gfCNCPoint2[27573] = {X 365.5713, Y 5.1234, Z -3.8333, A 0.000, B 0.000, C 0.000 }
gfCNCPoint2[27574] = {X 365.9457, Y 5.5507, Z -3.8333, A 0.000, B 0.000, C 0.000 }
gfCNCPoint2[27575] = {X 367.0655, Y 6.9489, Z -3.8333, A 0.000, B 0.000, C 0.000 }
gfCNCPoint2[27576] = {X 368.0925, Y 8.4166, Z -3.8333, A 0.000, B 0.000, C 0.000 }
gfCNCPoint2[27577] = {X 369.3414, Y 10.5295, Z -3.8333, A 0.000, B 0.000, C 0.000 }
gfCNCPoint2[27578] = {X 370.3982, Y 12.7448, Z -3.8333, A 0.000, B 0.000, C 0.000 }
gfCNCPoint2[27579] = {X 371.2546, Y 15.0450, Z -3.8333, A 0.000, B 0.000, C 0.000 }
gfCNCPoint2[27580] = {X 371.9038, Y 17.4120, Z -3.8333, A 0.000, B 0.000, C 0.000 }
gfCNCPoint2[27581] = {X 372.3604, Y 19.8116, Z -3.8333, A 0.000, B 0.000, C 0.000 }
gfCNCPoint2[27582] = {X 372.6464, Y 22.2374, Z -3.8333, A 0.000, B 0.000, C 0.000 }
gfCNCPoint2[27583] = {X 372.7605, Y 24.6774, Z -3.8333, A 0.000, B 0.000, C 0.000 }
gfCNCPoint2[27584] = {X 372.7020, Y 27.1193, Z -3.8333, A 0.000, B 0.000, C 0.000 }
gfCNCPoint2[27585] = {X 372.4713, Y 29.5510, Z -3.8333, A 0.000, B 0.000, C 0.000 }
gfCNCPoint2[27586] = {X 372.0694, Y 31.9603, Z -3.8333, A 0.000, B 0.000, C 0.000 }
gfCNCPoint2[27587] = {X 371.4833, Y 34.3147, Z -3.8333, A 0.000, B 0.000, C 0.000 }
gfCNCPoint2[27588] = {X 370.6918, Y 36.6082, Z -3.8333, A 0.000, B 0.000, C 0.000 }
gfCNCPoint2[27589] = {X 369.7011, Y 38.8229, Z -3.8333, A 0.000, B 0.000, C 0.000 }
gfCNCPoint2[27590] = {X 368.5189, Y 40.9417, Z -3.8333, A 0.000, B 0.000, C 0.000 }
gfCNCPoint2[27591] = {X 367.1545, Y 42.9479, Z -3.8333, A 0.000, B 0.000, C 0.000 }
gfCNCPoint2[27592] = {X 367.0324, Y 43.1153, Z -3.8333, A 0.000, B 0.000, C 0.000 }
gfCNCPoint2[27593] = {X 366.9645, Y 43.2035, Z -3.8333, A 0.000, B 0.000, C 0.000 }
gfCNCPoint2[27594] = {X 366.3182, Y 43.9969, Z -3.8333, A 0.000, B 0.000, C 0.000 }
gfCNCPoint2[27595] = {X 364.8822, Y 45.6080, Z -3.8333, A 0.000, B 0.000, C 0.000 }
gfCNCPoint2[27596] = {X 363.3086, Y 47.0851, Z -3.8333, A 0.000, B 0.000, C 0.000 }
gfCNCPoint2[27597] = {X 361.6099, Y 48.4164, Z -3.8333, A 0.000, B 0.000, C 0.000 }
gfCNCPoint2[27598] = {X 359.7996, Y 49.5915, Z -3.8333, A 0.000, B 0.000, C 0.000 }
gfCNCPoint2[27599] = {X 357.8920, Y 50.6010, Z -3.8333, A 0.000, B 0.000, C 0.000 }
gfCNCPoint2[27600] = {X 357.4593, Y 50.8059, Z -3.8333, A 0.000, B 0.000, C 0.000 }
gfCNCPoint2[27601] = {X 355.4789, Y 51.5741, Z -3.8333, A 0.000, B 0.000, C 0.000 }
gfCNCPoint2[27602] = {X 353.4424, Y 52.1780, Z -3.8333, A 0.000, B 0.000, C 0.000 }
gfCNCPoint2[27603] = {X 351.3633, Y 52.6134, Z -3.8333, A 0.000, B 0.000, C 0.000 }
gfCNCPoint2[27604] = {X 349.2556, Y 52.8775, Z -3.8333, A 0.000, B 0.000, C 0.000 }
gfCNCPoint2[27605] = {X 347.1333, Y 52.9685, Z -3.8333, A 0.000, B 0.000, C 0.000 }
gfCNCPoint2[27606] = {X 344.8131, Y 52.9262, Z -3.8333, A 0.000, B 0.000, C 0.000 }
gfCNCPoint2[27607] = {X 342.5052, Y 52.6831, Z -3.8333, A 0.000, B 0.000, C 0.000 }
gfCNCPoint2[27608] = {X 340.2271, Y 52.2410, Z -3.8333, A 0.000, B 0.000, C 0.000 }
gfCNCPoint2[27609] = {X 337.9959, Y 51.6033, Z -3.8333, A 0.000, B 0.000, C 0.000 }
gfCNCPoint2[27610] = {X 335.8282, Y 50.7746, Z -3.8333, A 0.000, B 0.000, C 0.000 }
gfCNCPoint2[27611] = {X 333.7405, Y 49.7614, Z -3.8333, A 0.000, B 0.000, C 0.000 }
gfCNCPoint2[27612] = {X 332.8345, Y 49.2281, Z -3.8333, A 0.000, B 0.000, C 0.000 }
gfCNCPoint2[27613] = {X 331.9502, Y 48.6598, Z -3.8333, A 0.000, B 0.000, C 0.000 }
gfCNCPoint2[27614] = {X 331.3028, Y 48.2115, Z -3.8333, A 0.000, B 0.000, C 0.000 }
gfCNCPoint2[27615] = {X 330.6689, Y 47.7445, Z -3.8333, A 0.000, B 0.000, C 0.000 }
gfCNCPoint2[27616] = {X 329.2171, Y 49.6556, Z -3.8333, A 0.000, B 0.000, C 0.000 }
gfCNCPoint2[27617] = {X 328.8724, Y 49.3896, Z -3.8333, A 0.000, B 0.000, C 0.000 }
gfCNCPoint2[27618] = {X 328.5317, Y 49.1186, Z -3.8333, A 0.000, B 0.000, C 0.000 }
gfCNCPoint2[27619] = {X 328.1266, Y 49.0390, Z -3.8333, A 0.000, B 0.000, C 0.000 }
gfCNCPoint2[27620] = {X 327.7253, Y 48.9423, Z -3.8333, A 0.000, B 0.000, C 0.000 }
gfCNCPoint2[27621] = {X 328.4864, Y 49.2670, Z -3.8333, A 0.000, B 0.000, C 0.000 }
gfCNCPoint2[27622] = {X 329.2171, Y 49.6556, Z -3.8333, A 0.000, B 0.000, C 0.000 }
gfCNCPoint2[27623] = {X 330.6689, Y 47.7445, Z -3.8333, A 0.000, B 0.000, C 0.000 }
gfCNCPoint2[27624] = {X 330.0951, Y 47.2962, Z -3.8333, A 0.000, B 0.000, C 0.000 }
gfCNCPoint2[27625] = {X 329.5337, Y 46.8324, Z -3.8333, A 0.000, B 0.000, C 0.000 }
gfCNCPoint2[27626] = {X 328.9312, Y 46.7520, Z -3.8333, A 0.000, B 0.000, C 0.000 }
gfCNCPoint2[27627] = {X 328.3374, Y 46.6216, Z -3.8333, A 0.000, B 0.000, C 0.000 }
gfCNCPoint2[27628] = {X 327.9789, Y 46.5172, Z -3.8333, A 0.000, B 0.000, C 0.000 }
gfCNCPoint2[27629] = {X 327.6263, Y 46.3944, Z -3.8333, A 0.000, B 0.000, C 0.000 }
gfCNCPoint2[27630] = {X 326.7320, Y 45.9864, Z -3.8333, A 0.000, B 0.000, C 0.000 }
gfCNCPoint2[27631] = {X 325.9009, Y 45.4616, Z -3.8333, A 0.000, B 0.000, C 0.000 }
gfCNCPoint2[27632] = {X 325.1480, Y 44.8296, Z -3.8333, A 0.000, B 0.000, C 0.000 }
gfCNCPoint2[27633] = {X 324.5140, Y 44.2115, Z -3.8333, A 0.000, B 0.000, C 0.000 }
gfCNCPoint2[27634] = {X 324.0475, Y 43.7117, Z -3.8333, A 0.000, B 0.000, C 0.000 }
gfCNCPoint2[27635] = {X 323.6300, Y 43.1703, Z -3.8333, A 0.000, B 0.000, C 0.000 }
gfCNCPoint2[27636] = {X 319.6957, Y 45.9200, Z -3.8333, A 0.000, B 0.000, C 0.000 }
gfCNCPoint2[27637] = {X 319.4780, Y 45.5976, Z -3.8333, A 0.000, B 0.000, C 0.000 }
gfCNCPoint2[27638] = {X 319.2708, Y 45.2683, Z -3.8333, A 0.000, B 0.000, C 0.000 }
gfCNCPoint2[27639] = {X 319.2514, Y 45.5948, Z -3.8333, A 0.000, B 0.000, C 0.000 }
gfCNCPoint2[27640] = {X 319.2174, Y 45.9200, Z -3.8333, A 0.000, B 0.000, C 0.000 }
gfCNCPoint2[27641] = {X 319.6957, Y 45.9200, Z -3.8333, A 0.000, B 0.000, C 0.000 }
gfCNCPoint2[27642] = {X 321.6628, Y 44.5452, Z -3.8333, A 0.000, B 0.000, C 0.000 }
gfCNCPoint2[27643] = {X 321.4884, Y 44.2868, Z -3.8333, A 0.000, B 0.000, C 0.000 }
gfCNCPoint2[27644] = {X 321.3224, Y 44.0230, Z -3.8333, A 0.000, B 0.000, C 0.000 }
gfCNCPoint2[27645] = {X 320.6712, Y 42.7455, Z -3.8333, A 0.000, B 0.000, C 0.000 }
gfCNCPoint2[27646] = {X 320.2158, Y 41.3859, Z -3.8333, A 0.000, B 0.000, C 0.000 }
gfCNCPoint2[27647] = {X 319.9663, Y 39.9740, Z -3.8333, A 0.000, B 0.000, C 0.000 }
gfCNCPoint2[27648] = {X 319.9281, Y 38.5406, Z -3.8333, A 0.000, B 0.000, C 0.000 }
gfCNCPoint2[27649] = {X 320.1020, Y 37.1174, Z -3.8333, A 0.000, B 0.000, C 0.000 }
gfCNCPoint2[27650] = {X 320.4301, Y 35.8909, Z -3.8333, A 0.000, B 0.000, C 0.000 }
gfCNCPoint2[27651] = {X 320.9158, Y 34.7180, Z -3.8333, A 0.000, B 0.000, C 0.000 }
gfCNCPoint2[27652] = {X 321.5508, Y 33.6186, Z -3.8333, A 0.000, B 0.000, C 0.000 }
gfCNCPoint2[27653] = {X 324.1378, Y 29.7505, Z -3.8333, A 0.000, B 0.000, C 0.000 }
gfCNCPoint2[27654] = {X 320.1479, Y 27.0821, Z -3.8333, A 0.000, B 0.000, C 0.000 }
gfCNCPoint2[27655] = {X 321.8042, Y 24.6057, Z -3.8333, A 0.000, B 0.000, C 0.000 }
gfCNCPoint2[27656] = {X 321.9898, Y 24.3356, Z -3.8333, A 0.000, B 0.000, C 0.000 }
gfCNCPoint2[27657] = {X 322.1814, Y 24.0697, Z -3.8333, A 0.000, B 0.000, C 0.000 }
gfCNCPoint2[27658] = {X 321.5380, Y 23.0772, Z -3.8333, A 0.000, B 0.000, C 0.000 }
gfCNCPoint2[27659] = {X 320.9777, Y 22.0354, Z -3.8333, A 0.000, B 0.000, C 0.000 }
gfCNCPoint2[27660] = {X 320.1480, Y 20.3286, Z -3.8333, A 0.000, B 0.000, C 0.000 }
gfCNCPoint2[27661] = {X 320.1479, Y 27.0821, Z -3.8333, A 0.000, B 0.000, C 0.000 }
gfCNCPoint2[27662] = {X 322.1429, Y 28.4163, Z -3.8333, A 0.000, B 0.000, C 0.000 }
gfCNCPoint2[27663] = {X 323.7975, Y 25.9423, Z -3.8333, A 0.000, B 0.000, C 0.000 }
gfCNCPoint2[27664] = {X 324.5112, Y 24.9841, Z -3.8333, A 0.000, B 0.000, C 0.000 }
gfCNCPoint2[27665] = {X 325.3162, Y 24.1010, Z -3.8333, A 0.000, B 0.000, C 0.000 }
gfCNCPoint2[27666] = {X 324.4812, Y 23.1413, Z -3.8333, A 0.000, B 0.000, C 0.000 }
gfCNCPoint2[27667] = {X 323.7518, Y 22.0990, Z -3.8333, A 0.000, B 0.000, C 0.000 }
gfCNCPoint2[27668] = {X 323.1360, Y 20.9859, Z -3.8333, A 0.000, B 0.000, C 0.000 }
gfCNCPoint2[27669] = {X 319.6151, Y 13.7428, Z -3.8333, A 0.000, B 0.000, C 0.000 }
gfCNCPoint2[27670] = {X 319.4387, Y 13.3633, Z -3.8333, A 0.000, B 0.000, C 0.000 }
gfCNCPoint2[27671] = {X 319.2755, Y 12.9779, Z -3.8333, A 0.000, B 0.000, C 0.000 }
gfCNCPoint2[27672] = {X 319.2755, Y 13.0353, Z -3.8333, A 0.000, B 0.000, C 0.000 }
gfCNCPoint2[27673] = {X 319.1698, Y 14.2156, Z -3.8333, A 0.000, B 0.000, C 0.000 }
gfCNCPoint2[27674] = {X 318.8739, Y 15.3632, Z -3.8333, A 0.000, B 0.000, C 0.000 }
gfCNCPoint2[27675] = {X 318.3958, Y 16.4476, Z -3.8333, A 0.000, B 0.000, C 0.000 }
gfCNCPoint2[27676] = {X 317.7480, Y 17.4400, Z -3.8333, A 0.000, B 0.000, C 0.000 }
gfCNCPoint2[27677] = {X 317.7478, Y 36.6506, Z -3.8333, A 0.000, B 0.000, C 0.000 }
gfCNCPoint2[27678] = {X 318.1572, Y 35.1201, Z -3.8333, A 0.000, B 0.000, C 0.000 }
gfCNCPoint2[27679] = {X 318.7634, Y 33.6563, Z -3.8333, A 0.000, B 0.000, C 0.000 }
gfCNCPoint2[27680] = {X 319.5559, Y 32.2844, Z -3.8333, A 0.000, B 0.000, C 0.000 }
gfCNCPoint2[27681] = {X 322.1429, Y 28.4163, Z -3.8333, A 0.000, B 0.000, C 0.000 }
gfCNCPoint2[27682] = {X 324.1378, Y 29.7505, Z -3.8333, A 0.000, B 0.000, C 0.000 }
gfCNCPoint2[27683] = {X 325.7908, Y 27.2790, Z -3.8333, A 0.000, B 0.000, C 0.000 }
gfCNCPoint2[27684] = {X 326.3627, Y 26.5111, Z -3.8333, A 0.000, B 0.000, C 0.000 }
gfCNCPoint2[27685] = {X 327.0077, Y 25.8035, Z -3.8333, A 0.000, B 0.000, C 0.000 }
gfCNCPoint2[27686] = {X 328.0707, Y 24.8904, Z -3.8333, A 0.000, B 0.000, C 0.000 }
gfCNCPoint2[27687] = {X 329.2543, Y 24.1403, Z -3.8333, A 0.000, B 0.000, C 0.000 }
gfCNCPoint2[27688] = {X 328.0859, Y 23.3667, Z -3.8333, A 0.000, B 0.000, C 0.000 }
gfCNCPoint2[27689] = {X 327.0414, Y 22.4326, Z -3.8333, A 0.000, B 0.000, C 0.000 }
gfCNCPoint2[27690] = {X 326.3723, Y 21.6635, Z -3.8333, A 0.000, B 0.000, C 0.000 }
gfCNCPoint2[27691] = {X 325.7878, Y 20.8284, Z -3.8333, A 0.000, B 0.000, C 0.000 }
gfCNCPoint2[27692] = {X 325.2944, Y 19.9364, Z -3.8333, A 0.000, B 0.000, C 0.000 }
gfCNCPoint2[27693] = {X 321.7736, Y 12.6936, Z -3.8333, A 0.000, B 0.000, C 0.000 }
gfCNCPoint2[27694] = {X 321.6322, Y 12.3894, Z -3.8333, A 0.000, B 0.000, C 0.000 }
gfCNCPoint2[27695] = {X 321.5015, Y 12.0806, Z -3.8333, A 0.000, B 0.000, C 0.000 }
gfCNCPoint2[27696] = {X 321.1058, Y 10.8774, Z -3.8333, A 0.000, B 0.000, C 0.000 }
gfCNCPoint2[27697] = {X 320.8706, Y 9.6327, Z -3.8333, A 0.000, B 0.000, C 0.000 }
gfCNCPoint2[27698] = {X 320.7999, Y 8.3681, Z -3.8333, A 0.000, B 0.000, C 0.000 }
gfCNCPoint2[27699] = {X 320.8950, Y 7.1050, Z -3.8333, A 0.000, B 0.000, C 0.000 }
gfCNCPoint2[27700] = {X 298.7842, Y 7.1050, Z -3.8333, A 0.000, B 0.000, C 0.000 }
gfCNCPoint2[27701] = {X 298.7842, Y 9.5050, Z -3.8333, A 0.000, B 0.000, C 0.000 }
gfCNCPoint2[27702] = {X 297.8292, Y 9.5050, Z -3.8333, A 0.000, B 0.000, C 0.000 }
gfCNCPoint2[27703] = {X 298.1371, Y 10.4755, Z -3.8333, A 0.000, B 0.000, C 0.000 }
gfCNCPoint2[27704] = {X 298.3067, Y 11.4795, Z -3.8333, A 0.000, B 0.000, C 0.000 }
gfCNCPoint2[27705] = {X 298.4762, Y 10.4755, Z -3.8333, A 0.000, B 0.000, C 0.000 }
gfCNCPoint2[27706] = {X 298.7842, Y 9.5050, Z -3.8333, A 0.000, B 0.000, C 0.000 }
gfCNCPoint2[27707] = {X 298.7842, Y 7.1050, Z -3.8333, A 0.000, B 0.000, C 0.000 }
gfCNCPoint2[27708] = {X 207.3611, Y 7.1050, Z -3.8333, A 0.000, B 0.000, C 0.000 }
gfCNCPoint2[27709] = {X 207.3611, Y 11.9050, Z -3.8333, A 0.000, B 0.000, C 0.000 }
gfCNCPoint2[27710] = {X 205.8559, Y 11.9050, Z -3.8333, A 0.000, B 0.000, C 0.000 }
gfCNCPoint2[27711] = {X 206.6109, Y 13.3410, Z -3.8333, A 0.000, B 0.000, C 0.000 }
gfCNCPoint2[27712] = {X 207.2366, Y 14.8379, Z -3.8333, A 0.000, B 0.000, C 0.000 }
gfCNCPoint2[27713] = {X 207.7977, Y 16.7110, Z -3.8333, A 0.000, B 0.000, C 0.000 }
gfCNCPoint2[27714] = {X 208.1767, Y 18.6291, Z -3.8333, A 0.000, B 0.000, C 0.000 }
gfCNCPoint2[27715] = {X 208.3702, Y 20.5748, Z -3.8333, A 0.000, B 0.000, C 0.000 }
gfCNCPoint2[27716] = {X 208.3763, Y 22.5301, Z -3.8333, A 0.000, B 0.000, C 0.000 }
gfCNCPoint2[27717] = {X 208.1951, Y 24.4769, Z -3.8333, A 0.000, B 0.000, C 0.000 }
gfCNCPoint2[27718] = {X 207.8282, Y 26.3974, Z -3.8333, A 0.000, B 0.000, C 0.000 }
gfCNCPoint2[27719] = {X 207.3612, Y 28.0098, Z -3.8333, A 0.000, B 0.000, C 0.000 }
gfCNCPoint2[27720] = {X 206.7379, Y 29.5684, Z -3.8333, A 0.000, B 0.000, C 0.000 }
gfCNCPoint2[27721] = {X 205.9643, Y 31.0582, Z -3.8333, A 0.000, B 0.000, C 0.000 }
gfCNCPoint2[27722] = {X 206.0464, Y 31.2164, Z -3.8333, A 0.000, B 0.000, C 0.000 }
gfCNCPoint2[27723] = {X 206.1255, Y 31.3761, Z -3.8333, A 0.000, B 0.000, C 0.000 }
gfCNCPoint2[27724] = {X 208.8852, Y 37.0775, Z -3.8333, A 0.000, B 0.000, C 0.000 }
gfCNCPoint2[27725] = {X 208.8852, Y 18.1982, Z -3.8333, A 0.000, B 0.000, C 0.000 }
gfCNCPoint2[27726] = {X 208.2331, Y 17.0021, Z -3.8333, A 0.000, B 0.000, C 0.000 }
gfCNCPoint2[27727] = {X 207.7553, Y 15.7263, Z -3.8333, A 0.000, B 0.000, C 0.000 }
gfCNCPoint2[27728] = {X 207.4614, Y 14.3961, Z -3.8333, A 0.000, B 0.000, C 0.000 }
gfCNCPoint2[27729] = {X 207.3572, Y 13.0378, Z -3.8333, A 0.000, B 0.000, C 0.000 }
gfCNCPoint2[27730] = {X 207.3570, Y 12.1868, Z -3.8333, A 0.000, B 0.000, C 0.000 }
gfCNCPoint2[27731] = {X 207.3580, Y 12.0459, Z -3.8333, A 0.000, B 0.000, C 0.000 }
gfCNCPoint2[27732] = {X 207.3611, Y 11.9050, Z -3.8333, A 0.000, B 0.000, C 0.000 }
gfCNCPoint2[27733] = {X 207.3611, Y 9.5050, Z -3.8333, A 0.000, B 0.000, C 0.000 }
gfCNCPoint2[27734] = {X 200.9069, Y 9.5050, Z -3.8333, A 0.000, B 0.000, C 0.000 }
gfCNCPoint2[27735] = {X 201.9803, Y 10.6137, Z -3.8333, A 0.000, B 0.000, C 0.000 }
gfCNCPoint2[27736] = {X 202.9419, Y 11.8206, Z -3.8333, A 0.000, B 0.000, C 0.000 }
gfCNCPoint2[27737] = {X 203.7829, Y 13.1145, Z -3.8333, A 0.000, B 0.000, C 0.000 }
gfCNCPoint2[27738] = {X 204.4363, Y 14.3564, Z -3.8333, A 0.000, B 0.000, C 0.000 }
gfCNCPoint2[27739] = {X 204.9784, Y 15.6507, Z -3.8333, A 0.000, B 0.000, C 0.000 }
gfCNCPoint2[27740] = {X 205.5510, Y 17.6374, Z -3.8333, A 0.000, B 0.000, C 0.000 }
gfCNCPoint2[27741] = {X 205.8919, Y 19.6767, Z -3.8333, A 0.000, B 0.000, C 0.000 }
gfCNCPoint2[27742] = {X 205.9964, Y 21.7416, Z -3.8333, A 0.000, B 0.000, C 0.000 }
gfCNCPoint2[27743] = {X 205.8631, Y 23.8049, Z -3.8333, A 0.000, B 0.000, C 0.000 }
gfCNCPoint2[27744] = {X 205.4940, Y 25.8393, Z -3.8333, A 0.000, B 0.000, C 0.000 }
gfCNCPoint2[27745] = {X 205.0929, Y 27.2255, Z -3.8333, A 0.000, B 0.000, C 0.000 }
gfCNCPoint2[27746] = {X 204.5574, Y 28.5655, Z -3.8333, A 0.000, B 0.000, C 0.000 }
gfCNCPoint2[27747] = {X 203.8927, Y 29.8464, Z -3.8333, A 0.000, B 0.000, C 0.000 }
gfCNCPoint2[27748] = {X 203.1052, Y 31.0557, Z -3.8333, A 0.000, B 0.000, C 0.000 }
gfCNCPoint2[27749] = {X 203.5732, Y 31.7148, Z -3.8333, A 0.000, B 0.000, C 0.000 }
gfCNCPoint2[27750] = {X 203.9653, Y 32.4217, Z -3.8333, A 0.000, B 0.000, C 0.000 }
gfCNCPoint2[27751] = {X 206.9865, Y 38.6634, Z -3.8333, A 0.000, B 0.000, C 0.000 }
gfCNCPoint2[27752] = {X 207.4240, Y 39.8017, Z -3.8333, A 0.000, B 0.000, C 0.000 }
gfCNCPoint2[27753] = {X 207.6653, Y 40.9971, Z -3.8333, A 0.000, B 0.000, C 0.000 }
gfCNCPoint2[27754] = {X 207.7038, Y 42.2159, Z -3.8333, A 0.000, B 0.000, C 0.000 }
gfCNCPoint2[27755] = {X 207.5382, Y 43.4241, Z -3.8333, A 0.000, B 0.000, C 0.000 }
gfCNCPoint2[27756] = {X 207.1733, Y 44.5877, Z -3.8333, A 0.000, B 0.000, C 0.000 }
gfCNCPoint2[27757] = {X 206.6193, Y 45.6741, Z -3.8333, A 0.000, B 0.000, C 0.000 }
gfCNCPoint2[27758] = {X 205.8917, Y 46.6527, Z -3.8333, A 0.000, B 0.000, C 0.000 }
gfCNCPoint2[27759] = {X 205.0110, Y 47.4962, Z -3.8333, A 0.000, B 0.000, C 0.000 }
gfCNCPoint2[27760] = {X 204.4738, Y 47.9305, Z -3.8333, A 0.000, B 0.000, C 0.000 }
gfCNCPoint2[27761] = {X 203.5892, Y 48.5431, Z -3.8333, A 0.000, B 0.000, C 0.000 }
gfCNCPoint2[27762] = {X 202.6241, Y 49.0188, Z -3.8333, A 0.000, B 0.000, C 0.000 }
gfCNCPoint2[27763] = {X 201.4895, Y 49.3730, Z -3.8333, A 0.000, B 0.000, C 0.000 }
gfCNCPoint2[27764] = {X 200.3125, Y 49.5382, Z -3.8333, A 0.000, B 0.000, C 0.000 }
gfCNCPoint2[27765] = {X 199.1243, Y 49.5100, Z -3.8333, A 0.000, B 0.000, C 0.000 }
gfCNCPoint2[27766] = {X 196.8333, Y 50.6067, Z -3.8333, A 0.000, B 0.000, C 0.000 }
gfCNCPoint2[27767] = {X 194.4618, Y 51.5162, Z -3.8333, A 0.000, B 0.000, C 0.000 }
gfCNCPoint2[27768] = {X 192.0250, Y 52.2327, Z -3.8333, A 0.000, B 0.000, C 0.000 }
gfCNCPoint2[27769] = {X 190.7221, Y 52.5183, Z -3.8333, A 0.000, B 0.000, C 0.000 }
gfCNCPoint2[27770] = {X 189.4061, Y 52.7356, Z -3.8333, A 0.000, B 0.000, C 0.000 }
gfCNCPoint2[27771] = {X 189.9005, Y 53.9113, Z -3.8333, A 0.000, B 0.000, C 0.000 }
gfCNCPoint2[27772] = {X 190.2683, Y 55.1326, Z -3.8333, A 0.000, B 0.000, C 0.000 }
gfCNCPoint2[27773] = {X 190.5269, Y 56.5560, Z -3.8333, A 0.000, B 0.000, C 0.000 }
gfCNCPoint2[27774] = {X 190.6135, Y 58.0000, Z -3.8333, A 0.000, B 0.000, C 0.000 }
gfCNCPoint2[27775] = {X 190.6132, Y 58.8767, Z -3.8333, A 0.000, B 0.000, C 0.000 }
gfCNCPoint2[27776] = {X 208.6252, Y 78.5345, Z -3.8333, A 0.000, B 0.000, C 0.000 }
gfCNCPoint2[27777] = {X 212.1642, Y 75.2918, Z -3.8333, A 0.000, B 0.000, C 0.000 }
gfCNCPoint2[27778] = {X 215.1994, Y 78.6043, Z -3.8333, A 0.000, B 0.000, C 0.000 }
gfCNCPoint2[27779] = {X 218.3280, Y 76.5999, Z -3.8333, A 0.000, B 0.000, C 0.000 }
gfCNCPoint2[27780] = {X 216.9962, Y 76.0772, Z -3.8333, A 0.000, B 0.000, C 0.000 }
gfCNCPoint2[27781] = {X 216.3765, Y 75.8848, Z -3.8333, A 0.000, B 0.000, C 0.000 }
gfCNCPoint2[27782] = {X 215.7328, Y 75.8035, Z -3.8333, A 0.000, B 0.000, C 0.000 }
gfCNCPoint2[27783] = {X 213.9348, Y 75.6432, Z -3.8333, A 0.000, B 0.000, C 0.000 }
gfCNCPoint2[27784] = {X 212.1642, Y 75.2918, Z -3.8333, A 0.000, B 0.000, C 0.000 }
gfCNCPoint2[27785] = {X 210.3947, Y 76.9131, Z -3.8333, A 0.000, B 0.000, C 0.000 }
gfCNCPoint2[27786] = {X 214.7939, Y 81.7143, Z -3.8333, A 0.000, B 0.000, C 0.000 }
gfCNCPoint2[27787] = {X 223.5827, Y 76.0838, Z -3.8333, A 0.000, B 0.000, C 0.000 }
gfCNCPoint2[27788] = {X 217.8854, Y 73.8480, Z -3.8333, A 0.000, B 0.000, C 0.000 }
gfCNCPoint2[27789] = {X 216.8722, Y 73.5366, Z -3.8333, A 0.000, B 0.000, C 0.000 }
gfCNCPoint2[27790] = {X 215.8204, Y 73.4051, Z -3.8333, A 0.000, B 0.000, C 0.000 }
gfCNCPoint2[27791] = {X 214.2768, Y 73.2676, Z -3.8333, A 0.000, B 0.000, C 0.000 }
gfCNCPoint2[27792] = {X 212.7566, Y 72.9660, Z -3.8333, A 0.000, B 0.000, C 0.000 }
gfCNCPoint2[27793] = {X 211.1575, Y 72.4584, Z -3.8333, A 0.000, B 0.000, C 0.000 }
gfCNCPoint2[27794] = {X 209.6279, Y 71.7692, Z -3.8333, A 0.000, B 0.000, C 0.000 }
gfCNCPoint2[27795] = {X 208.1882, Y 70.9078, Z -3.8333, A 0.000, B 0.000, C 0.000 }
gfCNCPoint2[27796] = {X 206.8579, Y 69.8855, Z -3.8333, A 0.000, B 0.000, C 0.000 }
gfCNCPoint2[27797] = {X 205.6547, Y 68.7163, Z -3.8333, A 0.000, B 0.000, C 0.000 }
gfCNCPoint2[27798] = {X 204.5949, Y 67.4157, Z -3.8333, A 0.000, B 0.000, C 0.000 }
gfCNCPoint2[27799] = {X 203.6926, Y 66.0013, Z -3.8333, A 0.000, B 0.000, C 0.000 }
gfCNCPoint2[27800] = {X 202.9600, Y 64.4920, Z -3.8333, A 0.000, B 0.000, C 0.000 }
gfCNCPoint2[27801] = {X 202.4068, Y 62.9081, Z -3.8333, A 0.000, B 0.000, C 0.000 }
gfCNCPoint2[27802] = {X 202.0406, Y 61.2709, Z -3.8333, A 0.000, B 0.000, C 0.000 }
gfCNCPoint2[27803] = {X 199.6721, Y 61.6582, Z -3.8333, A 0.000, B 0.000, C 0.000 }
gfCNCPoint2[27804] = {X 199.5095, Y 60.3402, Z -3.8333, A 0.000, B 0.000, C 0.000 }
gfCNCPoint2[27805] = {X 199.4510, Y 59.0136, Z -3.8333, A 0.000, B 0.000, C 0.000 }
gfCNCPoint2[27806] = {X 199.4508, Y 58.0000, Z -3.8333, A 0.000, B 0.000, C 0.000 }
gfCNCPoint2[27807] = {X 199.5412, Y 56.2556, Z -3.8333, A 0.000, B 0.000, C 0.000 }
gfCNCPoint2[27808] = {X 199.8114, Y 54.5298, Z -3.8333, A 0.000, B 0.000, C 0.000 }
gfCNCPoint2[27809] = {X 197.5977, Y 55.4810, Z -3.8333, A 0.000, B 0.000, C 0.000 }
gfCNCPoint2[27810] = {X 195.3260, Y 56.2839, Z -3.8333, A 0.000, B 0.000, C 0.000 }
gfCNCPoint2[27811] = {X 195.3578, Y 56.6300, Z -3.8333, A 0.000, B 0.000, C 0.000 }
gfCNCPoint2[27812] = {X 195.3825, Y 56.9766, Z -3.8333, A 0.000, B 0.000, C 0.000 }
gfCNCPoint2[27813] = {X 199.6721, Y 61.6582, Z -3.8333, A 0.000, B 0.000, C 0.000 }
gfCNCPoint2[27814] = {X 202.0406, Y 61.2709, Z -3.8333, A 0.000, B 0.000, C 0.000 }
gfCNCPoint2[27815] = {X 201.9013, Y 60.1428, Z -3.8333, A 0.000, B 0.000, C 0.000 }
gfCNCPoint2[27816] = {X 201.8510, Y 59.0073, Z -3.8333, A 0.000, B 0.000, C 0.000 }
gfCNCPoint2[27817] = {X 201.8508, Y 58.0000, Z -3.8333, A 0.000, B 0.000, C 0.000 }
gfCNCPoint2[27818] = {X 201.9283, Y 56.5036, Z -3.8333, A 0.000, B 0.000, C 0.000 }
gfCNCPoint2[27819] = {X 202.1601, Y 55.0232, Z -3.8333, A 0.000, B 0.000, C 0.000 }
gfCNCPoint2[27820] = {X 202.4969, Y 53.7230, Z -3.8333, A 0.000, B 0.000, C 0.000 }
gfCNCPoint2[27821] = {X 202.9527, Y 52.4596, Z -3.8333, A 0.000, B 0.000, C 0.000 }
gfCNCPoint2[27822] = {X 203.5236, Y 51.2439, Z -3.8333, A 0.000, B 0.000, C 0.000 }
gfCNCPoint2[27823] = {X 202.2637, Y 51.6554, Z -3.8333, A 0.000, B 0.000, C 0.000 }
gfCNCPoint2[27824] = {X 200.9594, Y 51.8913, Z -3.8333, A 0.000, B 0.000, C 0.000 }
gfCNCPoint2[27825] = {X 199.6352, Y 51.9470, Z -3.8333, A 0.000, B 0.000, C 0.000 }
gfCNCPoint2[27826] = {X 199.2148, Y 52.1550, Z -3.8333, A 0.000, B 0.000, C 0.000 }
gfCNCPoint2[27827] = {X 198.7916, Y 52.3572, Z -3.8333, A 0.000, B 0.000, C 0.000 }
gfCNCPoint2[27828] = {X 196.7764, Y 53.2250, Z -3.8333, A 0.000, B 0.000, C 0.000 }
gfCNCPoint2[27829] = {X 194.7096, Y 53.9612, Z -3.8333, A 0.000, B 0.000, C 0.000 }
gfCNCPoint2[27830] = {X 192.5997, Y 54.5629, Z -3.8333, A 0.000, B 0.000, C 0.000 }
gfCNCPoint2[27831] = {X 192.9063, Y 56.2411, Z -3.8333, A 0.000, B 0.000, C 0.000 }
gfCNCPoint2[27832] = {X 193.0134, Y 57.9437, Z -3.8333, A 0.000, B 0.000, C 0.000 }
gfCNCPoint2[27833] = {X 210.3947, Y 76.9131, Z -3.8333, A 0.000, B 0.000, C 0.000 }
gfCNCPoint2[27834] = {X 208.6252, Y 78.5345, Z -3.8333, A 0.000, B 0.000, C 0.000 }
gfCNCPoint2[27835] = {X 214.3884, Y 84.8243, Z -3.8333, A 0.000, B 0.000, C 0.000 }
gfCNCPoint2[27836] = {X 228.8373, Y 75.5678, Z -3.8333, A 0.000, B 0.000, C 0.000 }
gfCNCPoint2[27837] = {X 218.7726, Y 71.6180, Z -3.8333, A 0.000, B 0.000, C 0.000 }
gfCNCPoint2[27838] = {X 217.8432, Y 71.3042, Z -3.8333, A 0.000, B 0.000, C 0.000 }
gfCNCPoint2[27839] = {X 216.8839, Y 71.0995, Z -3.8333, A 0.000, B 0.000, C 0.000 }
gfCNCPoint2[27840] = {X 215.9073, Y 71.0066, Z -3.8333, A 0.000, B 0.000, C 0.000 }
gfCNCPoint2[27841] = {X 214.2374, Y 70.8313, Z -3.8333, A 0.000, B 0.000, C 0.000 }
gfCNCPoint2[27842] = {X 212.6079, Y 70.4261, Z -3.8333, A 0.000, B 0.000, C 0.000 }
gfCNCPoint2[27843] = {X 211.0503, Y 69.7988, Z -3.8333, A 0.000, B 0.000, C 0.000 }
gfCNCPoint2[27844] = {X 209.5948, Y 68.9617, Z -3.8333, A 0.000, B 0.000, C 0.000 }
gfCNCPoint2[27845] = {X 208.2694, Y 67.9308, Z -3.8333, A 0.000, B 0.000, C 0.000 }
gfCNCPoint2[27846] = {X 207.0998, Y 66.7260, Z -3.8333, A 0.000, B 0.000, C 0.000 }
gfCNCPoint2[27847] = {X 206.1085, Y 65.3707, Z -3.8333, A 0.000, B 0.000, C 0.000 }
gfCNCPoint2[27848] = {X 205.3147, Y 63.8911, Z -3.8333, A 0.000, B 0.000, C 0.000 }
gfCNCPoint2[27849] = {X 204.7338, Y 62.3157, Z -3.8333, A 0.000, B 0.000, C 0.000 }
gfCNCPoint2[27850] = {X 204.3769, Y 60.6749, Z -3.8333, A 0.000, B 0.000, C 0.000 }
gfCNCPoint2[27851] = {X 204.2510, Y 59.0005, Z -3.8333, A 0.000, B 0.000, C 0.000 }
gfCNCPoint2[27852] = {X 204.2508, Y 58.0000, Z -3.8333, A 0.000, B 0.000, C 0.000 }
gfCNCPoint2[27853] = {X 204.3397, Y 56.5376, Z -3.8333, A 0.000, B 0.000, C 0.000 }
gfCNCPoint2[27854] = {X 204.6049, Y 55.0967, Z -3.8333, A 0.000, B 0.000, C 0.000 }
gfCNCPoint2[27855] = {X 205.0426, Y 53.6986, Z -3.8333, A 0.000, B 0.000, C 0.000 }
gfCNCPoint2[27856] = {X 205.6463, Y 52.3637, Z -3.8333, A 0.000, B 0.000, C 0.000 }
gfCNCPoint2[27857] = {X 206.5298, Y 50.9383, Z -3.8333, A 0.000, B 0.000, C 0.000 }
gfCNCPoint2[27858] = {X 207.6022, Y 49.6491, Z -3.8333, A 0.000, B 0.000, C 0.000 }
gfCNCPoint2[27859] = {X 208.8428, Y 48.5208, Z -3.8333, A 0.000, B 0.000, C 0.000 }
gfCNCPoint2[27860] = {X 210.2277, Y 47.5751, Z -3.8333, A 0.000, B 0.000, C 0.000 }
gfCNCPoint2[27861] = {X 209.8801, Y 46.3328, Z -3.8333, A 0.000, B 0.000, C 0.000 }
gfCNCPoint2[27862] = {X 209.7572, Y 45.0487, Z -3.8333, A 0.000, B 0.000, C 0.000 }
gfCNCPoint2[27863] = {X 209.7570, Y 44.1967, Z -3.8333, A 0.000, B 0.000, C 0.000 }
gfCNCPoint2[27864] = {X 209.8559, Y 43.0066, Z -3.8333, A 0.000, B 0.000, C 0.000 }
gfCNCPoint2[27865] = {X 210.1498, Y 41.8492, Z -3.8333, A 0.000, B 0.000, C 0.000 }
gfCNCPoint2[27866] = {X 210.6306, Y 40.7561, Z -3.8333, A 0.000, B 0.000, C 0.000 }
gfCNCPoint2[27867] = {X 211.2852, Y 39.7574, Z -3.8333, A 0.000, B 0.000, C 0.000 }
gfCNCPoint2[27868] = {X 211.2852, Y 37.0775, Z -3.8333, A 0.000, B 0.000, C 0.000 }
gfCNCPoint2[27869] = {X 211.2849, Y 17.4403, Z -3.8333, A 0.000, B 0.000, C 0.000 }
gfCNCPoint2[27870] = {X 210.6364, Y 16.4465, Z -3.8333, A 0.000, B 0.000, C 0.000 }
gfCNCPoint2[27871] = {X 210.1579, Y 15.3605, Z -3.8333, A 0.000, B 0.000, C 0.000 }
gfCNCPoint2[27872] = {X 209.8622, Y 14.2112, Z -3.8333, A 0.000, B 0.000, C 0.000 }
gfCNCPoint2[27873] = {X 209.7572, Y 13.0291, Z -3.8333, A 0.000, B 0.000, C 0.000 }
gfCNCPoint2[27874] = {X 209.7570, Y 12.1868, Z -3.8333, A 0.000, B 0.000, C 0.000 }
gfCNCPoint2[27875] = {X 209.7578, Y 12.0808, Z -3.8333, A 0.000, B 0.000, C 0.000 }
gfCNCPoint2[27876] = {X 209.7601, Y 11.9749, Z -3.8333, A 0.000, B 0.000, C 0.000 }
gfCNCPoint2[27877] = {X 209.9068, Y 10.7177, Z -3.8333, A 0.000, B 0.000, C 0.000 }
gfCNCPoint2[27878] = {X 210.2690, Y 9.5050, Z -3.8333, A 0.000, B 0.000, C 0.000 }
gfCNCPoint2[27879] = {X 207.3611, Y 9.5050, Z -3.8333, A 0.000, B 0.000, C 0.000 }
gfCNCPoint2[27880] = {X 207.3611, Y 7.1050, Z -3.8333, A 0.000, B 0.000, C 0.000 }
gfCNCPoint2[27881] = {X 191.1443, Y 7.1050, Z -3.8333, A 0.000, B 0.000, C 0.000 }
gfCNCPoint2[27882] = {X 193.1012, Y 7.6483, Z -3.8333, A 0.000, B 0.000, C 0.000 }
gfCNCPoint2[27883] = {X 194.9845, Y 8.4084, Z -3.8333, A 0.000, B 0.000, C 0.000 }
gfCNCPoint2[27884] = {X 196.7702, Y 9.3758, Z -3.8333, A 0.000, B 0.000, C 0.000 }
gfCNCPoint2[27885] = {X 198.4355, Y 10.5381, Z -3.8333, A 0.000, B 0.000, C 0.000 }
gfCNCPoint2[27886] = {X 198.8575, Y 10.8885, Z -3.8333, A 0.000, B 0.000, C 0.000 }
gfCNCPoint2[27887] = {X 199.2650, Y 11.2555, Z -3.8333, A 0.000, B 0.000, C 0.000 }
gfCNCPoint2[27888] = {X 200.3500, Y 12.3982, Z -3.8333, A 0.000, B 0.000, C 0.000 }
gfCNCPoint2[27889] = {X 201.2956, Y 13.6586, Z -3.8333, A 0.000, B 0.000, C 0.000 }
gfCNCPoint2[27890] = {X 202.0892, Y 15.0198, Z -3.8333, A 0.000, B 0.000, C 0.000 }
gfCNCPoint2[27891] = {X 202.7202, Y 16.4636, Z -3.8333, A 0.000, B 0.000, C 0.000 }
gfCNCPoint2[27892] = {X 203.2139, Y 18.1834, Z -3.8333, A 0.000, B 0.000, C 0.000 }
gfCNCPoint2[27893] = {X 203.5072, Y 19.9484, Z -3.8333, A 0.000, B 0.000, C 0.000 }
gfCNCPoint2[27894] = {X 203.5963, Y 21.7354, Z -3.8333, A 0.000, B 0.000, C 0.000 }
gfCNCPoint2[27895] = {X 203.4800, Y 23.5208, Z -3.8333, A 0.000, B 0.000, C 0.000 }
gfCNCPoint2[27896] = {X 203.1598, Y 25.2812, Z -3.8333, A 0.000, B 0.000, C 0.000 }
gfCNCPoint2[27897] = {X 202.7594, Y 26.6265, Z -3.8333, A 0.000, B 0.000, C 0.000 }
gfCNCPoint2[27898] = {X 202.2078, Y 27.9173, Z -3.8333, A 0.000, B 0.000, C 0.000 }
gfCNCPoint2[27899] = {X 201.5122, Y 29.1365, Z -3.8333, A 0.000, B 0.000, C 0.000 }
gfCNCPoint2[27900] = {X 200.6817, Y 30.2681, Z -3.8333, A 0.000, B 0.000, C 0.000 }
gfCNCPoint2[27901] = {X 199.7272, Y 31.2973, Z -3.8333, A 0.000, B 0.000, C 0.000 }
gfCNCPoint2[27902] = {X 200.5668, Y 31.8698, Z -3.8333, A 0.000, B 0.000, C 0.000 }
gfCNCPoint2[27903] = {X 201.2695, Y 32.6038, Z -3.8333, A 0.000, B 0.000, C 0.000 }
gfCNCPoint2[27904] = {X 201.8050, Y 33.4674, Z -3.8333, A 0.000, B 0.000, C 0.000 }
gfCNCPoint2[27905] = {X 204.8262, Y 39.7091, Z -3.8333, A 0.000, B 0.000, C 0.000 }
gfCNCPoint2[27906] = {X 205.1508, Y 40.5847, Z -3.8333, A 0.000, B 0.000, C 0.000 }
gfCNCPoint2[27907] = {X 205.3026, Y 41.5062, Z -3.8333, A 0.000, B 0.000, C 0.000 }
gfCNCPoint2[27908] = {X 205.2761, Y 42.4397, Z -3.8333, A 0.000, B 0.000, C 0.000 }
gfCNCPoint2[27909] = {X 205.0723, Y 43.3511, Z -3.8333, A 0.000, B 0.000, C 0.000 }
gfCNCPoint2[27910] = {X 204.6986, Y 44.2070, Z -3.8333, A 0.000, B 0.000, C 0.000 }
gfCNCPoint2[27911] = {X 204.1687, Y 44.9760, Z -3.8333, A 0.000, B 0.000, C 0.000 }
gfCNCPoint2[27912] = {X 203.5020, Y 45.6299, Z -3.8333, A 0.000, B 0.000, C 0.000 }
gfCNCPoint2[27913] = {X 202.9657, Y 46.0636, Z -3.8333, A 0.000, B 0.000, C 0.000 }
gfCNCPoint2[27914] = {X 202.2136, Y 46.5639, Z -3.8333, A 0.000, B 0.000, C 0.000 }
gfCNCPoint2[27915] = {X 201.3824, Y 46.9175, Z -3.8333, A 0.000, B 0.000, C 0.000 }
gfCNCPoint2[27916] = {X 200.5003, Y 47.1123, Z -3.8333, A 0.000, B 0.000, C 0.000 }
gfCNCPoint2[27917] = {X 199.5975, Y 47.1416, Z -3.8333, A 0.000, B 0.000, C 0.000 }
gfCNCPoint2[27918] = {X 198.7046, Y 47.0045, Z -3.8333, A 0.000, B 0.000, C 0.000 }
gfCNCPoint2[27919] = {X 196.3903, Y 48.1789, Z -3.8333, A 0.000, B 0.000, C 0.000 }
gfCNCPoint2[27920] = {X 193.9811, Y 49.1437, Z -3.8333, A 0.000, B 0.000, C 0.000 }
gfCNCPoint2[27921] = {X 191.4959, Y 49.8913, Z -3.8333, A 0.000, B 0.000, C 0.000 }
gfCNCPoint2[27922] = {X 190.2926, Y 50.1569, Z -3.8333, A 0.000, B 0.000, C 0.000 }
gfCNCPoint2[27923] = {X 189.0769, Y 50.3583, Z -3.8333, A 0.000, B 0.000, C 0.000 }
gfCNCPoint2[27924] = {X 186.8985, Y 50.5559, Z -3.8333, A 0.000, B 0.000, C 0.000 }
gfCNCPoint2[27925] = {X 184.7112, Y 50.5476, Z -3.8333, A 0.000, B 0.000, C 0.000 }
gfCNCPoint2[27926] = {X 184.7356, Y 50.0682, Z -3.8333, A 0.000, B 0.000, C 0.000 }
gfCNCPoint2[27927] = {X 183.1153, Y 49.9273, Z -3.8333, A 0.000, B 0.000, C 0.000 }
gfCNCPoint2[27928] = {X 181.5093, Y 49.6709, Z -3.8333, A 0.000, B 0.000, C 0.000 }
gfCNCPoint2[27929] = {X 179.6141, Y 49.1972, Z -3.8333, A 0.000, B 0.000, C 0.000 }
gfCNCPoint2[27930] = {X 177.7853, Y 48.5105, Z -3.8333, A 0.000, B 0.000, C 0.000 }
gfCNCPoint2[27931] = {X 176.0466, Y 47.6200, Z -3.8333, A 0.000, B 0.000, C 0.000 }
gfCNCPoint2[27932] = {X 174.4207, Y 46.5371, Z -3.8333, A 0.000, B 0.000, C 0.000 }
gfCNCPoint2[27933] = {X 173.1806, Y 45.4904, Z -3.8333, A 0.000, B 0.000, C 0.000 }
gfCNCPoint2[27934] = {X 172.0771, Y 44.3007, Z -3.8333, A 0.000, B 0.000, C 0.000 }
gfCNCPoint2[27935] = {X 171.1264, Y 42.9855, Z -3.8333, A 0.000, B 0.000, C 0.000 }
gfCNCPoint2[27936] = {X 170.3428, Y 41.5644, Z -3.8333, A 0.000, B 0.000, C 0.000 }
gfCNCPoint2[27937] = {X 169.7379, Y 40.0586, Z -3.8333, A 0.000, B 0.000, C 0.000 }
gfCNCPoint2[27938] = {X 169.3206, Y 38.4904, Z -3.8333, A 0.000, B 0.000, C 0.000 }
gfCNCPoint2[27939] = {X 169.0973, Y 36.8830, Z -3.8333, A 0.000, B 0.000, C 0.000 }
gfCNCPoint2[27940] = {X 169.0129, Y 35.0393, Z -3.8333, A 0.000, B 0.000, C 0.000 }
gfCNCPoint2[27941] = {X 169.1600, Y 33.1996, Z -3.8333, A 0.000, B 0.000, C 0.000 }
gfCNCPoint2[27942] = {X 169.5362, Y 31.3927, Z -3.8333, A 0.000, B 0.000, C 0.000 }
gfCNCPoint2[27943] = {X 170.1356, Y 29.6472, Z -3.8333, A 0.000, B 0.000, C 0.000 }
gfCNCPoint2[27944] = {X 170.7627, Y 28.3595, Z -3.8333, A 0.000, B 0.000, C 0.000 }
gfCNCPoint2[27945] = {X 171.5526, Y 27.1648, Z -3.8333, A 0.000, B 0.000, C 0.000 }
gfCNCPoint2[27946] = {X 172.4918, Y 26.0836, Z -3.8333, A 0.000, B 0.000, C 0.000 }
gfCNCPoint2[27947] = {X 173.5642, Y 25.1342, Z -3.8333, A 0.000, B 0.000, C 0.000 }
gfCNCPoint2[27948] = {X 174.7514, Y 24.3331, Z -3.8333, A 0.000, B 0.000, C 0.000 }
gfCNCPoint2[27949] = {X 173.9912, Y 23.9228, Z -3.8333, A 0.000, B 0.000, C 0.000 }
gfCNCPoint2[27950] = {X 173.3259, Y 23.3719, Z -3.8333, A 0.000, B 0.000, C 0.000 }
gfCNCPoint2[27951] = {X 172.7810, Y 22.7016, Z -3.8333, A 0.000, B 0.000, C 0.000 }
gfCNCPoint2[27952] = {X 172.3776, Y 21.9378, Z -3.8333, A 0.000, B 0.000, C 0.000 }
gfCNCPoint2[27953] = {X 169.7664, Y 15.5423, Z -3.8333, A 0.000, B 0.000, C 0.000 }
gfCNCPoint2[27954] = {X 169.5125, Y 14.6752, Z -3.8333, A 0.000, B 0.000, C 0.000 }
gfCNCPoint2[27955] = {X 169.4412, Y 13.7745, Z -3.8333, A 0.000, B 0.000, C 0.000 }
gfCNCPoint2[27956] = {X 169.5553, Y 12.8782, Z -3.8333, A 0.000, B 0.000, C 0.000 }
gfCNCPoint2[27957] = {X 169.8501, Y 12.0241, Z -3.8333, A 0.000, B 0.000, C 0.000 }
gfCNCPoint2[27958] = {X 170.3131, Y 11.2482, Z -3.8333, A 0.000, B 0.000, C 0.000 }
gfCNCPoint2[27959] = {X 170.9249, Y 10.5833, Z -3.8333, A 0.000, B 0.000, C 0.000 }
gfCNCPoint2[27960] = {X 171.6596, Y 10.0573, Z -3.8333, A 0.000, B 0.000, C 0.000 }
gfCNCPoint2[27961] = {X 172.2916, Y 9.6970, Z -3.8333, A 0.000, B 0.000, C 0.000 }
gfCNCPoint2[27962] = {X 173.1812, Y 9.3215, Z -3.8333, A 0.000, B 0.000, C 0.000 }
gfCNCPoint2[27963] = {X 174.1312, Y 9.1491, Z -3.8333, A 0.000, B 0.000, C 0.000 }
gfCNCPoint2[27964] = {X 175.0960, Y 9.1881, Z -3.8333, A 0.000, B 0.000, C 0.000 }
gfCNCPoint2[27965] = {X 176.0290, Y 9.4366, Z -3.8333, A 0.000, B 0.000, C 0.000 }
gfCNCPoint2[27966] = {X 178.2250, Y 8.5159, Z -3.8333, A 0.000, B 0.000, C 0.000 }
gfCNCPoint2[27967] = {X 180.5019, Y 7.8190, Z -3.8333, A 0.000, B 0.000, C 0.000 }
gfCNCPoint2[27968] = {X 182.8370, Y 7.3528, Z -3.8333, A 0.000, B 0.000, C 0.000 }
gfCNCPoint2[27969] = {X 185.2069, Y 7.1220, Z -3.8333, A 0.000, B 0.000, C 0.000 }
gfCNCPoint2[27970] = {X 187.5881, Y 7.1288, Z -3.8333, A 0.000, B 0.000, C 0.000 }
gfCNCPoint2[27971] = {X 189.9567, Y 7.3733, Z -3.8333, A 0.000, B 0.000, C 0.000 }
gfCNCPoint2[27972] = {X 191.7226, Y 7.7364, Z -3.8333, A 0.000, B 0.000, C 0.000 }
gfCNCPoint2[27973] = {X 193.4418, Y 8.2791, Z -3.8333, A 0.000, B 0.000, C 0.000 }
gfCNCPoint2[27974] = {X 195.0963, Y 8.9955, Z -3.8333, A 0.000, B 0.000, C 0.000 }
gfCNCPoint2[27975] = {X 196.6683, Y 9.8781, Z -3.8333, A 0.000, B 0.000, C 0.000 }
gfCNCPoint2[27976] = {X 198.1414, Y 10.9175, Z -3.8333, A 0.000, B 0.000, C 0.000 }
gfCNCPoint2[27977] = {X 199.2077, Y 11.8672, Z -3.8333, A 0.000, B 0.000, C 0.000 }
gfCNCPoint2[27978] = {X 200.1645, Y 12.9271, Z -3.8333, A 0.000, B 0.000, C 0.000 }
gfCNCPoint2[27979] = {X 201.0005, Y 14.0847, Z -3.8333, A 0.000, B 0.000, C 0.000 }
gfCNCPoint2[27980] = {X 201.7060, Y 15.3261, Z -3.8333, A 0.000, B 0.000, C 0.000 }
gfCNCPoint2[27981] = {X 202.2724, Y 16.6369, Z -3.8333, A 0.000, B 0.000, C 0.000 }
gfCNCPoint2[27982] = {X 202.7486, Y 18.3014, Z -3.8333, A 0.000, B 0.000, C 0.000 }
gfCNCPoint2[27983] = {X 203.0311, Y 20.0095, Z -3.8333, A 0.000, B 0.000, C 0.000 }
gfCNCPoint2[27984] = {X 203.1163, Y 21.7387, Z -3.8333, A 0.000, B 0.000, C 0.000 }
gfCNCPoint2[27985] = {X 203.0031, Y 23.4663, Z -3.8333, A 0.000, B 0.000, C 0.000 }
gfCNCPoint2[27986] = {X 202.6929, Y 25.1696, Z -3.8333, A 0.000, B 0.000, C 0.000 }
gfCNCPoint2[27987] = {X 202.2583, Y 26.5986, Z -3.8333, A 0.000, B 0.000, C 0.000 }
gfCNCPoint2[27988] = {X 201.6461, Y 27.9610, Z -3.8333, A 0.000, B 0.000, C 0.000 }
gfCNCPoint2[27989] = {X 200.8664, Y 29.2350, Z -3.8333, A 0.000, B 0.000, C 0.000 }
gfCNCPoint2[27990] = {X 199.9317, Y 30.4000, Z -3.8333, A 0.000, B 0.000, C 0.000 }
gfCNCPoint2[27991] = {X 198.8569, Y 31.4373, Z -3.8333, A 0.000, B 0.000, C 0.000 }
gfCNCPoint2[27992] = {X 199.6401, Y 31.7990, Z -3.8333, A 0.000, B 0.000, C 0.000 }
gfCNCPoint2[27993] = {X 200.3377, Y 32.3066, Z -3.8333, A 0.000, B 0.000, C 0.000 }
gfCNCPoint2[27994] = {X 200.9228, Y 32.9405, Z -3.8333, A 0.000, B 0.000, C 0.000 }
gfCNCPoint2[27995] = {X 201.3730, Y 33.6764, Z -3.8333, A 0.000, B 0.000, C 0.000 }
gfCNCPoint2[27996] = {X 204.3942, Y 39.9182, Z -3.8333, A 0.000, B 0.000, C 0.000 }
gfCNCPoint2[27997] = {X 204.7207, Y 40.8441, Z -3.8333, A 0.000, B 0.000, C 0.000 }
gfCNCPoint2[27998] = {X 204.8337, Y 41.8194, Z -3.8333, A 0.000, B 0.000, C 0.000 }
gfCNCPoint2[27999] = {X 204.7276, Y 42.7955, Z -3.8333, A 0.000, B 0.000, C 0.000 }
gfCNCPoint2[28000] = {X 204.4078, Y 43.7238, Z -3.8333, A 0.000, B 0.000, C 0.000 }
gfCNCPoint2[28001] = {X 203.8900, Y 44.5580, Z -3.8333, A 0.000, B 0.000, C 0.000 }
gfCNCPoint2[28002] = {X 203.2002, Y 45.2567, Z -3.8333, A 0.000, B 0.000, C 0.000 }
gfCNCPoint2[28003] = {X 202.6639, Y 45.6903, Z -3.8333, A 0.000, B 0.000, C 0.000 }
gfCNCPoint2[28004] = {X 201.9524, Y 46.1592, Z -3.8333, A 0.000, B 0.000, C 0.000 }
gfCNCPoint2[28005] = {X 201.1640, Y 46.4827, Z -3.8333, A 0.000, B 0.000, C 0.000 }
gfCNCPoint2[28006] = {X 200.3282, Y 46.6486, Z -3.8333, A 0.000, B 0.000, C 0.000 }
gfCNCPoint2[28007] = {X 199.4761, Y 46.6509, Z -3.8333, A 0.000, B 0.000, C 0.000 }
gfCNCPoint2[28008] = {X 198.6394, Y 46.4893, Z -3.8333, A 0.000, B 0.000, C 0.000 }
gfCNCPoint2[28009] = {X 196.3110, Y 47.6876, Z -3.8333, A 0.000, B 0.000, C 0.000 }
gfCNCPoint2[28010] = {X 193.8833, Y 48.6693, Z -3.8333, A 0.000, B 0.000, C 0.000 }
gfCNCPoint2[28011] = {X 191.3765, Y 49.4264, Z -3.8333, A 0.000, B 0.000, C 0.000 }
gfCNCPoint2[28012] = {X 189.1875, Y 49.8577, Z -3.8333, A 0.000, B 0.000, C 0.000 }
gfCNCPoint2[28013] = {X 186.9667, Y 50.0723, Z -3.8333, A 0.000, B 0.000, C 0.000 }
gfCNCPoint2[28014] = {X 184.7356, Y 50.0682, Z -3.8333, A 0.000, B 0.000, C 0.000 }
gfCNCPoint2[28015] = {X 184.7112, Y 50.5476, Z -3.8333, A 0.000, B 0.000, C 0.000 }
gfCNCPoint2[28016] = {X 185.7074, Y 51.5010, Z -3.8333, A 0.000, B 0.000, C 0.000 }
gfCNCPoint2[28017] = {X 186.5581, Y 52.5863, Z -3.8333, A 0.000, B 0.000, C 0.000 }
gfCNCPoint2[28018] = {X 187.2459, Y 53.7815, Z -3.8333, A 0.000, B 0.000, C 0.000 }
gfCNCPoint2[28019] = {X 187.7794, Y 55.1337, Z -3.8333, A 0.000, B 0.000, C 0.000 }
gfCNCPoint2[28020] = {X 188.1044, Y 56.5505, Z -3.8333, A 0.000, B 0.000, C 0.000 }
gfCNCPoint2[28021] = {X 188.2135, Y 58.0000, Z -3.8333, A 0.000, B 0.000, C 0.000 }
gfCNCPoint2[28022] = {X 188.2132, Y 59.0140, Z -3.8333, A 0.000, B 0.000, C 0.000 }
gfCNCPoint2[28023] = {X 188.2026, Y 59.3928, Z -3.8333, A 0.000, B 0.000, C 0.000 }
gfCNCPoint2[28024] = {X 188.1773, Y 59.7708, Z -3.8333, A 0.000, B 0.000, C 0.000 }
gfCNCPoint2[28025] = {X 213.5228, Y 87.4322, Z -3.8333, A 0.000, B 0.000, C 0.000 }
gfCNCPoint2[28026] = {X 214.2178, Y 87.3797, Z -3.8333, A 0.000, B 0.000, C 0.000 }
gfCNCPoint2[28027] = {X 214.9136, Y 87.3382, Z -3.8333, A 0.000, B 0.000, C 0.000 }
gfCNCPoint2[28028] = {X 234.0920, Y 75.0517, Z -3.8333, A 0.000, B 0.000, C 0.000 }
gfCNCPoint2[28029] = {X 219.6585, Y 69.3875, Z -3.8333, A 0.000, B 0.000, C 0.000 }
gfCNCPoint2[28030] = {X 218.4696, Y 68.9874, Z -3.8333, A 0.000, B 0.000, C 0.000 }
gfCNCPoint2[28031] = {X 217.2426, Y 68.7265, Z -3.8333, A 0.000, B 0.000, C 0.000 }
gfCNCPoint2[28032] = {X 215.9937, Y 68.6082, Z -3.8333, A 0.000, B 0.000, C 0.000 }
gfCNCPoint2[28033] = {X 214.5234, Y 68.4438, Z -3.8333, A 0.000, B 0.000, C 0.000 }
gfCNCPoint2[28034] = {X 213.0953, Y 68.0573, Z -3.8333, A 0.000, B 0.000, C 0.000 }
gfCNCPoint2[28035] = {X 211.7428, Y 67.4577, Z -3.8333, A 0.000, B 0.000, C 0.000 }
gfCNCPoint2[28036] = {X 210.4974, Y 66.6590, Z -3.8333, A 0.000, B 0.000, C 0.000 }
gfCNCPoint2[28037] = {X 209.3883, Y 65.6798, Z -3.8333, A 0.000, B 0.000, C 0.000 }
gfCNCPoint2[28038] = {X 208.4414, Y 64.5430, Z -3.8333, A 0.000, B 0.000, C 0.000 }
gfCNCPoint2[28039] = {X 207.6788, Y 63.2752, Z -3.8333, A 0.000, B 0.000, C 0.000 }
gfCNCPoint2[28040] = {X 207.1183, Y 61.9060, Z -3.8333, A 0.000, B 0.000, C 0.000 }
gfCNCPoint2[28041] = {X 206.7730, Y 60.4674, Z -3.8333, A 0.000, B 0.000, C 0.000 }
gfCNCPoint2[28042] = {X 206.6510, Y 58.9930, Z -3.8333, A 0.000, B 0.000, C 0.000 }
gfCNCPoint2[28043] = {X 206.6508, Y 58.0000, Z -3.8333, A 0.000, B 0.000, C 0.000 }
gfCNCPoint2[28044] = {X 206.7577, Y 56.5655, Z -3.8333, A 0.000, B 0.000, C 0.000 }
gfCNCPoint2[28045] = {X 207.0760, Y 55.1628, Z -3.8333, A 0.000, B 0.000, C 0.000 }
gfCNCPoint2[28046] = {X 207.5986, Y 53.8226, Z -3.8333, A 0.000, B 0.000, C 0.000 }
gfCNCPoint2[28047] = {X 208.3140, Y 52.5747, Z -3.8333, A 0.000, B 0.000, C 0.000 }
gfCNCPoint2[28048] = {X 209.2065, Y 51.4466, Z -3.8333, A 0.000, B 0.000, C 0.000 }
gfCNCPoint2[28049] = {X 210.2563, Y 50.4632, Z -3.8333, A 0.000, B 0.000, C 0.000 }
gfCNCPoint2[28050] = {X 211.4402, Y 49.6463, Z -3.8333, A 0.000, B 0.000, C 0.000 }
gfCNCPoint2[28051] = {X 212.5893, Y 49.0723, Z -3.8333, A 0.000, B 0.000, C 0.000 }
gfCNCPoint2[28052] = {X 213.8042, Y 48.6556, Z -3.8333, A 0.000, B 0.000, C 0.000 }
gfCNCPoint2[28053] = {X 213.2578, Y 48.0874, Z -3.8333, A 0.000, B 0.000, C 0.000 }
gfCNCPoint2[28054] = {X 212.8100, Y 47.4386, Z -3.8333, A 0.000, B 0.000, C 0.000 }
gfCNCPoint2[28055] = {X 212.4725, Y 46.7262, Z -3.8333, A 0.000, B 0.000, C 0.000 }
gfCNCPoint2[28056] = {X 212.2401, Y 45.8965, Z -3.8333, A 0.000, B 0.000, C 0.000 }
gfCNCPoint2[28057] = {X 212.1572, Y 45.0389, Z -3.8333, A 0.000, B 0.000, C 0.000 }
gfCNCPoint2[28058] = {X 212.1570, Y 44.1967, Z -3.8333, A 0.000, B 0.000, C 0.000 }
gfCNCPoint2[28059] = {X 212.2383, Y 43.3157, Z -3.8333, A 0.000, B 0.000, C 0.000 }
gfCNCPoint2[28060] = {X 212.4796, Y 42.4646, Z -3.8333, A 0.000, B 0.000, C 0.000 }
gfCNCPoint2[28061] = {X 212.8725, Y 41.6719, Z -3.8333, A 0.000, B 0.000, C 0.000 }
gfCNCPoint2[28062] = {X 213.4040, Y 40.9647, Z -3.8333, A 0.000, B 0.000, C 0.000 }
gfCNCPoint2[28063] = {X 213.6825, Y 40.6575, Z -3.8333, A 0.000, B 0.000, C 0.000 }
gfCNCPoint2[28064] = {X 213.6852, Y 40.3041, Z -3.8333, A 0.000, B 0.000, C 0.000 }
gfCNCPoint2[28065] = {X 213.6852, Y 17.4645, Z -3.8333, A 0.000, B 0.000, C 0.000 }
gfCNCPoint2[28066] = {X 213.6799, Y 16.7697, Z -3.8333, A 0.000, B 0.000, C 0.000 }
gfCNCPoint2[28067] = {X 213.6796, Y 16.5195, Z -3.8333, A 0.000, B 0.000, C 0.000 }
gfCNCPoint2[28068] = {X 213.0403, Y 15.7782, Z -3.8333, A 0.000, B 0.000, C 0.000 }
gfCNCPoint2[28069] = {X 212.5619, Y 14.9242, Z -3.8333, A 0.000, B 0.000, C 0.000 }
gfCNCPoint2[28070] = {X 212.2635, Y 13.9919, Z -3.8333, A 0.000, B 0.000, C 0.000 }
gfCNCPoint2[28071] = {X 212.1572, Y 13.0188, Z -3.8333, A 0.000, B 0.000, C 0.000 }
gfCNCPoint2[28072] = {X 212.1570, Y 12.1868, Z -3.8333, A 0.000, B 0.000, C 0.000 }
gfCNCPoint2[28073] = {X 212.2436, Y 11.2717, Z -3.8333, A 0.000, B 0.000, C 0.000 }
gfCNCPoint2[28074] = {X 212.5002, Y 10.3891, Z -3.8333, A 0.000, B 0.000, C 0.000 }
gfCNCPoint2[28075] = {X 212.9449, Y 9.5280, Z -3.8333, A 0.000, B 0.000, C 0.000 }
gfCNCPoint2[28076] = {X 213.5510, Y 8.7718, Z -3.8333, A 0.000, B 0.000, C 0.000 }
gfCNCPoint2[28077] = {X 214.2946, Y 8.1503, Z -3.8333, A 0.000, B 0.000, C 0.000 }
gfCNCPoint2[28078] = {X 215.1464, Y 7.6879, Z -3.8333, A 0.000, B 0.000, C 0.000 }
gfCNCPoint2[28079] = {X 216.0727, Y 7.4030, Z -3.8333, A 0.000, B 0.000, C 0.000 }
gfCNCPoint2[28080] = {X 217.0370, Y 7.3068, Z -3.8333, A 0.000, B 0.000, C 0.000 }
gfCNCPoint2[28081] = {X 223.4805, Y 7.3068, Z -3.8333, A 0.000, B 0.000, C 0.000 }
gfCNCPoint2[28082] = {X 224.4448, Y 7.4030, Z -3.8333, A 0.000, B 0.000, C 0.000 }
gfCNCPoint2[28083] = {X 225.3711, Y 7.6879, Z -3.8333, A 0.000, B 0.000, C 0.000 }
gfCNCPoint2[28084] = {X 226.2229, Y 8.1503, Z -3.8333, A 0.000, B 0.000, C 0.000 }
gfCNCPoint2[28085] = {X 226.9665, Y 8.7718, Z -3.8333, A 0.000, B 0.000, C 0.000 }
gfCNCPoint2[28086] = {X 227.5726, Y 9.5280, Z -3.8333, A 0.000, B 0.000, C 0.000 }
gfCNCPoint2[28087] = {X 228.0173, Y 10.3891, Z -3.8333, A 0.000, B 0.000, C 0.000 }
gfCNCPoint2[28088] = {X 228.2739, Y 11.2717, Z -3.8333, A 0.000, B 0.000, C 0.000 }
gfCNCPoint2[28089] = {X 228.3605, Y 12.1868, Z -3.8333, A 0.000, B 0.000, C 0.000 }
gfCNCPoint2[28090] = {X 228.3603, Y 13.0237, Z -3.8333, A 0.000, B 0.000, C 0.000 }
gfCNCPoint2[28091] = {X 228.2529, Y 13.9972, Z -3.8333, A 0.000, B 0.000, C 0.000 }
gfCNCPoint2[28092] = {X 227.9533, Y 14.9296, Z -3.8333, A 0.000, B 0.000, C 0.000 }
gfCNCPoint2[28093] = {X 227.4735, Y 15.7834, Z -3.8333, A 0.000, B 0.000, C 0.000 }
gfCNCPoint2[28094] = {X 226.8330, Y 16.5242, Z -3.8333, A 0.000, B 0.000, C 0.000 }
gfCNCPoint2[28095] = {X 226.8333, Y 25.8483, Z -3.8333, A 0.000, B 0.000, C 0.000 }
gfCNCPoint2[28096] = {X 231.6333, Y 25.8481, Z -3.8333, A 0.000, B 0.000, C 0.000 }
gfCNCPoint2[28097] = {X 231.6338, Y 38.9909, Z -3.8333, A 0.000, B 0.000, C 0.000 }
gfCNCPoint2[28098] = {X 231.6440, Y 39.0069, Z -3.8333, A 0.000, B 0.000, C 0.000 }
gfCNCPoint2[28099] = {X 232.3931, Y 37.9855, Z -3.8333, A 0.000, B 0.000, C 0.000 }
gfCNCPoint2[28100] = {X 233.2692, Y 37.0706, Z -3.8333, A 0.000, B 0.000, C 0.000 }
gfCNCPoint2[28101] = {X 234.2573, Y 36.2780, Z -3.8333, A 0.000, B 0.000, C 0.000 }
gfCNCPoint2[28102] = {X 235.5694, Y 33.7097, Z -3.8333, A 0.000, B 0.000, C 0.000 }
gfCNCPoint2[28103] = {X 234.4287, Y 32.2855, Z -3.8333, A 0.000, B 0.000, C 0.000 }
gfCNCPoint2[28104] = {X 233.4504, Y 30.7451, Z -3.8333, A 0.000, B 0.000, C 0.000 }
gfCNCPoint2[28105] = {X 232.6462, Y 29.1072, Z -3.8333, A 0.000, B 0.000, C 0.000 }
gfCNCPoint2[28106] = {X 232.0258, Y 27.3911, Z -3.8333, A 0.000, B 0.000, C 0.000 }
gfCNCPoint2[28107] = {X 231.8155, Y 26.6232, Z -3.8333, A 0.000, B 0.000, C 0.000 }
gfCNCPoint2[28108] = {X 231.6333, Y 25.8481, Z -3.8333, A 0.000, B 0.000, C 0.000 }
gfCNCPoint2[28109] = {X 229.2333, Y 25.8482, Z -3.8333, A 0.000, B 0.000, C 0.000 }
gfCNCPoint2[28110] = {X 229.2338, Y 39.7481, Z -3.8333, A 0.000, B 0.000, C 0.000 }
gfCNCPoint2[28111] = {X 229.4332, Y 40.0179, Z -3.8333, A 0.000, B 0.000, C 0.000 }
gfCNCPoint2[28112] = {X 229.6200, Y 40.2966, Z -3.8333, A 0.000, B 0.000, C 0.000 }
gfCNCPoint2[28113] = {X 230.1055, Y 41.1910, Z -3.8333, A 0.000, B 0.000, C 0.000 }
gfCNCPoint2[28114] = {X 230.4616, Y 42.1443, Z -3.8333, A 0.000, B 0.000, C 0.000 }
gfCNCPoint2[28115] = {X 230.6813, Y 43.1379, Z -3.8333, A 0.000, B 0.000, C 0.000 }
gfCNCPoint2[28116] = {X 230.7603, Y 44.1524, Z -3.8333, A 0.000, B 0.000, C 0.000 }
gfCNCPoint2[28117] = {X 230.7605, Y 45.0000, Z -3.8333, A 0.000, B 0.000, C 0.000 }
gfCNCPoint2[28118] = {X 230.7459, Y 45.4609, Z -3.8333, A 0.000, B 0.000, C 0.000 }
gfCNCPoint2[28119] = {X 230.7021, Y 45.9200, Z -3.8333, A 0.000, B 0.000, C 0.000 }
gfCNCPoint2[28120] = {X 232.5859, Y 45.9200, Z -3.8333, A 0.000, B 0.000, C 0.000 }
gfCNCPoint2[28121] = {X 232.5421, Y 45.4609, Z -3.8333, A 0.000, B 0.000, C 0.000 }
gfCNCPoint2[28122] = {X 232.5275, Y 45.0000, Z -3.8333, A 0.000, B 0.000, C 0.000 }
gfCNCPoint2[28123] = {X 232.5275, Y 44.2090, Z -3.8333, A 0.000, B 0.000, C 0.000 }
gfCNCPoint2[28124] = {X 232.6006, Y 43.1798, Z -3.8333, A 0.000, B 0.000, C 0.000 }
gfCNCPoint2[28125] = {X 232.8184, Y 42.1714, Z -3.8333, A 0.000, B 0.000, C 0.000 }
gfCNCPoint2[28126] = {X 233.1766, Y 41.2038, Z -3.8333, A 0.000, B 0.000, C 0.000 }
gfCNCPoint2[28127] = {X 233.6680, Y 40.2966, Z -3.8333, A 0.000, B 0.000, C 0.000 }
gfCNCPoint2[28128] = {X 234.3527, Y 39.3876, Z -3.8333, A 0.000, B 0.000, C 0.000 }
gfCNCPoint2[28129] = {X 235.1707, Y 38.5964, Z -3.8333, A 0.000, B 0.000, C 0.000 }
gfCNCPoint2[28130] = {X 236.1021, Y 37.9424, Z -3.8333, A 0.000, B 0.000, C 0.000 }
gfCNCPoint2[28131] = {X 238.5000, Y 33.2486, Z -3.8333, A 0.000, B 0.000, C 0.000 }
gfCNCPoint2[28132] = {X 237.3863, Y 32.1409, Z -3.8333, A 0.000, B 0.000, C 0.000 }
gfCNCPoint2[28133] = {X 236.4010, Y 30.9175, Z -3.8333, A 0.000, B 0.000, C 0.000 }
gfCNCPoint2[28134] = {X 235.5560, Y 29.5932, Z -3.8333, A 0.000, B 0.000, C 0.000 }
gfCNCPoint2[28135] = {X 234.8617, Y 28.1842, Z -3.8333, A 0.000, B 0.000, C 0.000 }
gfCNCPoint2[28136] = {X 234.3264, Y 26.7074, Z -3.8333, A 0.000, B 0.000, C 0.000 }
gfCNCPoint2[28137] = {X 234.1404, Y 26.0275, Z -3.8333, A 0.000, B 0.000, C 0.000 }
gfCNCPoint2[28138] = {X 233.9792, Y 25.3414, Z -3.8333, A 0.000, B 0.000, C 0.000 }
gfCNCPoint2[28139] = {X 233.6675, Y 23.4533, Z -3.8333, A 0.000, B 0.000, C 0.000 }
gfCNCPoint2[28140] = {X 233.5423, Y 21.5437, Z -3.8333, A 0.000, B 0.000, C 0.000 }
gfCNCPoint2[28141] = {X 233.6051, Y 19.6310, Z -3.8333, A 0.000, B 0.000, C 0.000 }
gfCNCPoint2[28142] = {X 233.8550, Y 17.7337, Z -3.8333, A 0.000, B 0.000, C 0.000 }
gfCNCPoint2[28143] = {X 234.2897, Y 15.8700, Z -3.8333, A 0.000, B 0.000, C 0.000 }
gfCNCPoint2[28144] = {X 234.7355, Y 14.5427, Z -3.8333, A 0.000, B 0.000, C 0.000 }
gfCNCPoint2[28145] = {X 235.3047, Y 13.2635, Z -3.8333, A 0.000, B 0.000, C 0.000 }
gfCNCPoint2[28146] = {X 233.1605, Y 12.1853, Z -3.8333, A 0.000, B 0.000, C 0.000 }
gfCNCPoint2[28147] = {X 233.2319, Y 12.0448, Z -3.8333, A 0.000, B 0.000, C 0.000 }
gfCNCPoint2[28148] = {X 233.3047, Y 11.9050, Z -3.8333, A 0.000, B 0.000, C 0.000 }
gfCNCPoint2[28149] = {X 233.1564, Y 11.9050, Z -3.8333, A 0.000, B 0.000, C 0.000 }
gfCNCPoint2[28150] = {X 233.1594, Y 12.0452, Z -3.8333, A 0.000, B 0.000, C 0.000 }
gfCNCPoint2[28151] = {X 233.1605, Y 12.1853, Z -3.8333, A 0.000, B 0.000, C 0.000 }
gfCNCPoint2[28152] = {X 235.3047, Y 13.2635, Z -3.8333, A 0.000, B 0.000, C 0.000 }
gfCNCPoint2[28153] = {X 235.3662, Y 13.1426, Z -3.8333, A 0.000, B 0.000, C 0.000 }
gfCNCPoint2[28154] = {X 235.4288, Y 13.0223, Z -3.8333, A 0.000, B 0.000, C 0.000 }
gfCNCPoint2[28155] = {X 236.1701, Y 11.7671, Z -3.8333, A 0.000, B 0.000, C 0.000 }
gfCNCPoint2[28156] = {X 237.0312, Y 10.5909, Z -3.8333, A 0.000, B 0.000, C 0.000 }
gfCNCPoint2[28157] = {X 238.0038, Y 9.5050, Z -3.8333, A 0.000, B 0.000, C 0.000 }
gfCNCPoint2[28158] = {X 230.2485, Y 9.5050, Z -3.8333, A 0.000, B 0.000, C 0.000 }
gfCNCPoint2[28159] = {X 230.6107, Y 10.7177, Z -3.8333, A 0.000, B 0.000, C 0.000 }
gfCNCPoint2[28160] = {X 230.7574, Y 11.9749, Z -3.8333, A 0.000, B 0.000, C 0.000 }
gfCNCPoint2[28161] = {X 230.7597, Y 12.0808, Z -3.8333, A 0.000, B 0.000, C 0.000 }
gfCNCPoint2[28162] = {X 230.7605, Y 12.1868, Z -3.8333, A 0.000, B 0.000, C 0.000 }
gfCNCPoint2[28163] = {X 230.7602, Y 13.0462, Z -3.8333, A 0.000, B 0.000, C 0.000 }
gfCNCPoint2[28164] = {X 230.6531, Y 14.2236, Z -3.8333, A 0.000, B 0.000, C 0.000 }
gfCNCPoint2[28165] = {X 230.3569, Y 15.3682, Z -3.8333, A 0.000, B 0.000, C 0.000 }
gfCNCPoint2[28166] = {X 229.8793, Y 16.4498, Z -3.8333, A 0.000, B 0.000, C 0.000 }
gfCNCPoint2[28167] = {X 229.2330, Y 17.4398, Z -3.8333, A 0.000, B 0.000, C 0.000 }
gfCNCPoint2[28168] = {X 229.2333, Y 25.8482, Z -3.8333, A 0.000, B 0.000, C 0.000 }
gfCNCPoint2[28169] = {X 226.8333, Y 25.8483, Z -3.8333, A 0.000, B 0.000, C 0.000 }
gfCNCPoint2[28170] = {X 226.8338, Y 40.6635, Z -3.8333, A 0.000, B 0.000, C 0.000 }
gfCNCPoint2[28171] = {X 227.4742, Y 41.4043, Z -3.8333, A 0.000, B 0.000, C 0.000 }
gfCNCPoint2[28172] = {X 227.9537, Y 42.2581, Z -3.8333, A 0.000, B 0.000, C 0.000 }
gfCNCPoint2[28173] = {X 228.2530, Y 43.1905, Z -3.8333, A 0.000, B 0.000, C 0.000 }
gfCNCPoint2[28174] = {X 228.3603, Y 44.1638, Z -3.8333, A 0.000, B 0.000, C 0.000 }
gfCNCPoint2[28175] = {X 228.3605, Y 45.0000, Z -3.8333, A 0.000, B 0.000, C 0.000 }
gfCNCPoint2[28176] = {X 228.3507, Y 45.3090, Z -3.8333, A 0.000, B 0.000, C 0.000 }
gfCNCPoint2[28177] = {X 228.3214, Y 45.6167, Z -3.8333, A 0.000, B 0.000, C 0.000 }
gfCNCPoint2[28178] = {X 228.0910, Y 46.5992, Z -3.8333, A 0.000, B 0.000, C 0.000 }
gfCNCPoint2[28179] = {X 227.6635, Y 47.5134, Z -3.8333, A 0.000, B 0.000, C 0.000 }
gfCNCPoint2[28180] = {X 227.0571, Y 48.3200, Z -3.8333, A 0.000, B 0.000, C 0.000 }
gfCNCPoint2[28181] = {X 226.7053, Y 47.9934, Z -3.8333, A 0.000, B 0.000, C 0.000 }
gfCNCPoint2[28182] = {X 226.0261, Y 48.5889, Z -3.8333, A 0.000, B 0.000, C 0.000 }
gfCNCPoint2[28183] = {X 225.2396, Y 49.0331, Z -3.8333, A 0.000, B 0.000, C 0.000 }
gfCNCPoint2[28184] = {X 224.3790, Y 49.3073, Z -3.8333, A 0.000, B 0.000, C 0.000 }
gfCNCPoint2[28185] = {X 223.4805, Y 49.4000, Z -3.8333, A 0.000, B 0.000, C 0.000 }
gfCNCPoint2[28186] = {X 217.0370, Y 49.4000, Z -3.8333, A 0.000, B 0.000, C 0.000 }
gfCNCPoint2[28187] = {X 216.0579, Y 49.2897, Z -3.8333, A 0.000, B 0.000, C 0.000 }
gfCNCPoint2[28188] = {X 215.1279, Y 48.9643, Z -3.8333, A 0.000, B 0.000, C 0.000 }
gfCNCPoint2[28189] = {X 214.2936, Y 48.4400, Z -3.8333, A 0.000, B 0.000, C 0.000 }
gfCNCPoint2[28190] = {X 213.5969, Y 47.7433, Z -3.8333, A 0.000, B 0.000, C 0.000 }
gfCNCPoint2[28191] = {X 213.0727, Y 46.9091, Z -3.8333, A 0.000, B 0.000, C 0.000 }
gfCNCPoint2[28192] = {X 212.7473, Y 45.9791, Z -3.8333, A 0.000, B 0.000, C 0.000 }
gfCNCPoint2[28193] = {X 212.6370, Y 45.0000, Z -3.8333, A 0.000, B 0.000, C 0.000 }
gfCNCPoint2[28194] = {X 212.6370, Y 44.1967, Z -3.8333, A 0.000, B 0.000, C 0.000 }
gfCNCPoint2[28195] = {X 212.7102, Y 43.4036, Z -3.8333, A 0.000, B 0.000, C 0.000 }
gfCNCPoint2[28196] = {X 212.9274, Y 42.6373, Z -3.8333, A 0.000, B 0.000, C 0.000 }
gfCNCPoint2[28197] = {X 213.2812, Y 41.9238, Z -3.8333, A 0.000, B 0.000, C 0.000 }
gfCNCPoint2[28198] = {X 213.7596, Y 41.2871, Z -3.8333, A 0.000, B 0.000, C 0.000 }
gfCNCPoint2[28199] = {X 214.1611, Y 40.8442, Z -3.8333, A 0.000, B 0.000, C 0.000 }
gfCNCPoint2[28200] = {X 214.1652, Y 40.3060, Z -3.8333, A 0.000, B 0.000, C 0.000 }
gfCNCPoint2[28201] = {X 214.1652, Y 17.4626, Z -3.8333, A 0.000, B 0.000, C 0.000 }
gfCNCPoint2[28202] = {X 214.1599, Y 16.7692, Z -3.8333, A 0.000, B 0.000, C 0.000 }
gfCNCPoint2[28203] = {X 214.1594, Y 16.3066, Z -3.8333, A 0.000, B 0.000, C 0.000 }
gfCNCPoint2[28204] = {X 213.5168, Y 15.6178, Z -3.8333, A 0.000, B 0.000, C 0.000 }
gfCNCPoint2[28205] = {X 213.0356, Y 14.8081, Z -3.8333, A 0.000, B 0.000, C 0.000 }
gfCNCPoint2[28206] = {X 212.7378, Y 13.9145, Z -3.8333, A 0.000, B 0.000, C 0.000 }
gfCNCPoint2[28207] = {X 212.6370, Y 12.9779, Z -3.8333, A 0.000, B 0.000, C 0.000 }
gfCNCPoint2[28208] = {X 212.6370, Y 12.1868, Z -3.8333, A 0.000, B 0.000, C 0.000 }
gfCNCPoint2[28209] = {X 212.7473, Y 11.2077, Z -3.8333, A 0.000, B 0.000, C 0.000 }
gfCNCPoint2[28210] = {X 213.0728, Y 10.2777, Z -3.8333, A 0.000, B 0.000, C 0.000 }
gfCNCPoint2[28211] = {X 213.5970, Y 9.4435, Z -3.8333, A 0.000, B 0.000, C 0.000 }
gfCNCPoint2[28212] = {X 214.2937, Y 8.7468, Z -3.8333, A 0.000, B 0.000, C 0.000 }
gfCNCPoint2[28213] = {X 215.1279, Y 8.2226, Z -3.8333, A 0.000, B 0.000, C 0.000 }
gfCNCPoint2[28214] = {X 216.0579, Y 7.8971, Z -3.8333, A 0.000, B 0.000, C 0.000 }
gfCNCPoint2[28215] = {X 217.0370, Y 7.7868, Z -3.8333, A 0.000, B 0.000, C 0.000 }
gfCNCPoint2[28216] = {X 223.4805, Y 7.7868, Z -3.8333, A 0.000, B 0.000, C 0.000 }
gfCNCPoint2[28217] = {X 224.4596, Y 7.8971, Z -3.8333, A 0.000, B 0.000, C 0.000 }
gfCNCPoint2[28218] = {X 225.3896, Y 8.2226, Z -3.8333, A 0.000, B 0.000, C 0.000 }
gfCNCPoint2[28219] = {X 226.2238, Y 8.7468, Z -3.8333, A 0.000, B 0.000, C 0.000 }
gfCNCPoint2[28220] = {X 226.9205, Y 9.4435, Z -3.8333, A 0.000, B 0.000, C 0.000 }
gfCNCPoint2[28221] = {X 227.4447, Y 10.2777, Z -3.8333, A 0.000, B 0.000, C 0.000 }
gfCNCPoint2[28222] = {X 227.7702, Y 11.2077, Z -3.8333, A 0.000, B 0.000, C 0.000 }
gfCNCPoint2[28223] = {X 227.8805, Y 12.1868, Z -3.8333, A 0.000, B 0.000, C 0.000 }
gfCNCPoint2[28224] = {X 227.8802, Y 13.0233, Z -3.8333, A 0.000, B 0.000, C 0.000 }
gfCNCPoint2[28225] = {X 227.7719, Y 13.9493, Z -3.8333, A 0.000, B 0.000, C 0.000 }
gfCNCPoint2[28226] = {X 227.4709, Y 14.8318, Z -3.8333, A 0.000, B 0.000, C 0.000 }
gfCNCPoint2[28227] = {X 226.9907, Y 15.6310, Z -3.8333, A 0.000, B 0.000, C 0.000 }
gfCNCPoint2[28228] = {X 226.3529, Y 16.3110, Z -3.8333, A 0.000, B 0.000, C 0.000 }
gfCNCPoint2[28229] = {X 226.3539, Y 40.8766, Z -3.8333, A 0.000, B 0.000, C 0.000 }
gfCNCPoint2[28230] = {X 226.9981, Y 41.5656, Z -3.8333, A 0.000, B 0.000, C 0.000 }
gfCNCPoint2[28231] = {X 227.4807, Y 42.3762, Z -3.8333, A 0.000, B 0.000, C 0.000 }
gfCNCPoint2[28232] = {X 227.7794, Y 43.2710, Z -3.8333, A 0.000, B 0.000, C 0.000 }
gfCNCPoint2[28233] = {X 227.8805, Y 44.2089, Z -3.8333, A 0.000, B 0.000, C 0.000 }
gfCNCPoint2[28234] = {X 227.8805, Y 45.0000, Z -3.8333, A 0.000, B 0.000, C 0.000 }
gfCNCPoint2[28235] = {X 227.8037, Y 45.8182, Z -3.8333, A 0.000, B 0.000, C 0.000 }
gfCNCPoint2[28236] = {X 227.5762, Y 46.6079, Z -3.8333, A 0.000, B 0.000, C 0.000 }
gfCNCPoint2[28237] = {X 227.2057, Y 47.3415, Z -3.8333, A 0.000, B 0.000, C 0.000 }
gfCNCPoint2[28238] = {X 226.7053, Y 47.9934, Z -3.8333, A 0.000, B 0.000, C 0.000 }
gfCNCPoint2[28239] = {X 227.0571, Y 48.3200, Z -3.8333, A 0.000, B 0.000, C 0.000 }
gfCNCPoint2[28240] = {X 236.2309, Y 48.3200, Z -3.8333, A 0.000, B 0.000, C 0.000 }
gfCNCPoint2[28241] = {X 235.6245, Y 47.5134, Z -3.8333, A 0.000, B 0.000, C 0.000 }
gfCNCPoint2[28242] = {X 235.1970, Y 46.5992, Z -3.8333, A 0.000, B 0.000, C 0.000 }
gfCNCPoint2[28243] = {X 234.9666, Y 45.6167, Z -3.8333, A 0.000, B 0.000, C 0.000 }
gfCNCPoint2[28244] = {X 234.9373, Y 45.3090, Z -3.8333, A 0.000, B 0.000, C 0.000 }
gfCNCPoint2[28245] = {X 234.9275, Y 45.0000, Z -3.8333, A 0.000, B 0.000, C 0.000 }
gfCNCPoint2[28246] = {X 234.9275, Y 44.2089, Z -3.8333, A 0.000, B 0.000, C 0.000 }
gfCNCPoint2[28247] = {X 235.0194, Y 43.2661, Z -3.8333, A 0.000, B 0.000, C 0.000 }
gfCNCPoint2[28248] = {X 235.2917, Y 42.3588, Z -3.8333, A 0.000, B 0.000, C 0.000 }
gfCNCPoint2[28249] = {X 235.7342, Y 41.5212, Z -3.8333, A 0.000, B 0.000, C 0.000 }
gfCNCPoint2[28250] = {X 236.3302, Y 40.7849, Z -3.8333, A 0.000, B 0.000, C 0.000 }
gfCNCPoint2[28251] = {X 237.0572, Y 40.1776, Z -3.8333, A 0.000, B 0.000, C 0.000 }
gfCNCPoint2[28252] = {X 237.8878, Y 39.7222, Z -3.8333, A 0.000, B 0.000, C 0.000 }
gfCNCPoint2[28253] = {X 241.5465, Y 32.5608, Z -3.8333, A 0.000, B 0.000, C 0.000 }
gfCNCPoint2[28254] = {X 240.2120, Y 31.5582, Z -3.8333, A 0.000, B 0.000, C 0.000 }
gfCNCPoint2[28255] = {X 239.0313, Y 30.3783, Z -3.8333, A 0.000, B 0.000, C 0.000 }
gfCNCPoint2[28256] = {X 238.0276, Y 29.0446, Z -3.8333, A 0.000, B 0.000, C 0.000 }
gfCNCPoint2[28257] = {X 237.2208, Y 27.5834, Z -3.8333, A 0.000, B 0.000, C 0.000 }
gfCNCPoint2[28258] = {X 236.6269, Y 26.0234, Z -3.8333, A 0.000, B 0.000, C 0.000 }
gfCNCPoint2[28259] = {X 236.1917, Y 24.1498, Z -3.8333, A 0.000, B 0.000, C 0.000 }
gfCNCPoint2[28260] = {X 235.9698, Y 22.2392, Z -3.8333, A 0.000, B 0.000, C 0.000 }
gfCNCPoint2[28261] = {X 235.9640, Y 20.3157, Z -3.8333, A 0.000, B 0.000, C 0.000 }
gfCNCPoint2[28262] = {X 236.1742, Y 18.4037, Z -3.8333, A 0.000, B 0.000, C 0.000 }
gfCNCPoint2[28263] = {X 236.5979, Y 16.5275, Z -3.8333, A 0.000, B 0.000, C 0.000 }
gfCNCPoint2[28264] = {X 237.1172, Y 15.0569, Z -3.8333, A 0.000, B 0.000, C 0.000 }
gfCNCPoint2[28265] = {X 237.8169, Y 13.6631, Z -3.8333, A 0.000, B 0.000, C 0.000 }
gfCNCPoint2[28266] = {X 238.6859, Y 12.3681, Z -3.8333, A 0.000, B 0.000, C 0.000 }
gfCNCPoint2[28267] = {X 239.7105, Y 11.1924, Z -3.8333, A 0.000, B 0.000, C 0.000 }
gfCNCPoint2[28268] = {X 240.8748, Y 10.1542, Z -3.8333, A 0.000, B 0.000, C 0.000 }
gfCNCPoint2[28269] = {X 242.1601, Y 9.2704, Z -3.8333, A 0.000, B 0.000, C 0.000 }
gfCNCPoint2[28270] = {X 243.5462, Y 8.5548, Z -3.8333, A 0.000, B 0.000, C 0.000 }
gfCNCPoint2[28271] = {X 245.0110, Y 8.0188, Z -3.8333, A 0.000, B 0.000, C 0.000 }
gfCNCPoint2[28272] = {X 246.5316, Y 7.6708, Z -3.8333, A 0.000, B 0.000, C 0.000 }
gfCNCPoint2[28273] = {X 248.6761, Y 7.3933, Z -3.8333, A 0.000, B 0.000, C 0.000 }
gfCNCPoint2[28274] = {X 250.8369, Y 7.3109, Z -3.8333, A 0.000, B 0.000, C 0.000 }
gfCNCPoint2[28275] = {X 266.7608, Y 7.3109, Z -3.8333, A 0.000, B 0.000, C 0.000 }
gfCNCPoint2[28276] = {X 267.7190, Y 7.4123, Z -3.8333, A 0.000, B 0.000, C 0.000 }
gfCNCPoint2[28277] = {X 268.6387, Y 7.7000, Z -3.8333, A 0.000, B 0.000, C 0.000 }
gfCNCPoint2[28278] = {X 269.4840, Y 8.1627, Z -3.8333, A 0.000, B 0.000, C 0.000 }
gfCNCPoint2[28279] = {X 270.2219, Y 8.7823, Z -3.8333, A 0.000, B 0.000, C 0.000 }
gfCNCPoint2[28280] = {X 270.8238, Y 9.5349, Z -3.8333, A 0.000, B 0.000, C 0.000 }
gfCNCPoint2[28281] = {X 271.2662, Y 10.3910, Z -3.8333, A 0.000, B 0.000, C 0.000 }
gfCNCPoint2[28282] = {X 271.5233, Y 11.2719, Z -3.8333, A 0.000, B 0.000, C 0.000 }
gfCNCPoint2[28283] = {X 271.6110, Y 12.1855, Z -3.8333, A 0.000, B 0.000, C 0.000 }
gfCNCPoint2[28284] = {X 271.6108, Y 13.0237, Z -3.8333, A 0.000, B 0.000, C 0.000 }
gfCNCPoint2[28285] = {X 271.5128, Y 13.9524, Z -3.8333, A 0.000, B 0.000, C 0.000 }
gfCNCPoint2[28286] = {X 271.2396, Y 14.8453, Z -3.8333, A 0.000, B 0.000, C 0.000 }
gfCNCPoint2[28287] = {X 275.6743, Y 16.6820, Z -3.8333, A 0.000, B 0.000, C 0.000 }
gfCNCPoint2[28288] = {X 275.3125, Y 17.4569, Z -3.8333, A 0.000, B 0.000, C 0.000 }
gfCNCPoint2[28289] = {X 274.8837, Y 18.1968, Z -3.8333, A 0.000, B 0.000, C 0.000 }
gfCNCPoint2[28290] = {X 274.8836, Y 38.9897, Z -3.8333, A 0.000, B 0.000, C 0.000 }
gfCNCPoint2[28291] = {X 275.3139, Y 39.7326, Z -3.8333, A 0.000, B 0.000, C 0.000 }
gfCNCPoint2[28292] = {X 275.6768, Y 40.5107, Z -3.8333, A 0.000, B 0.000, C 0.000 }
gfCNCPoint2[28293] = {X 276.0379, Y 39.7361, Z -3.8333, A 0.000, B 0.000, C 0.000 }
gfCNCPoint2[28294] = {X 276.4656, Y 38.9962, Z -3.8333, A 0.000, B 0.000, C 0.000 }
gfCNCPoint2[28295] = {X 276.4652, Y 18.1972, Z -3.8333, A 0.000, B 0.000, C 0.000 }
gfCNCPoint2[28296] = {X 276.0363, Y 17.4571, Z -3.8333, A 0.000, B 0.000, C 0.000 }
gfCNCPoint2[28297] = {X 275.6743, Y 16.6820, Z -3.8333, A 0.000, B 0.000, C 0.000 }
gfCNCPoint2[28298] = {X 273.4570, Y 15.7637, Z -3.8333, A 0.000, B 0.000, C 0.000 }
gfCNCPoint2[28299] = {X 273.0264, Y 16.6341, Z -3.8333, A 0.000, B 0.000, C 0.000 }
gfCNCPoint2[28300] = {X 272.4837, Y 17.4395, Z -3.8333, A 0.000, B 0.000, C 0.000 }
gfCNCPoint2[28301] = {X 272.4836, Y 39.7471, Z -3.8333, A 0.000, B 0.000, C 0.000 }
gfCNCPoint2[28302] = {X 273.0275, Y 40.5547, Z -3.8333, A 0.000, B 0.000, C 0.000 }
gfCNCPoint2[28303] = {X 273.4588, Y 41.4276, Z -3.8333, A 0.000, B 0.000, C 0.000 }
gfCNCPoint2[28304] = {X 273.7589, Y 42.3096, Z -3.8333, A 0.000, B 0.000, C 0.000 }
gfCNCPoint2[28305] = {X 273.9439, Y 43.2226, Z -3.8333, A 0.000, B 0.000, C 0.000 }
gfCNCPoint2[28306] = {X 274.0108, Y 44.1519, Z -3.8333, A 0.000, B 0.000, C 0.000 }
gfCNCPoint2[28307] = {X 274.0110, Y 45.0000, Z -3.8333, A 0.000, B 0.000, C 0.000 }
gfCNCPoint2[28308] = {X 273.9884, Y 45.5734, Z -3.8333, A 0.000, B 0.000, C 0.000 }
gfCNCPoint2[28309] = {X 273.9207, Y 46.1433, Z -3.8333, A 0.000, B 0.000, C 0.000 }
gfCNCPoint2[28310] = {X 275.0713, Y 45.9760, Z -3.8333, A 0.000, B 0.000, C 0.000 }
gfCNCPoint2[28311] = {X 276.2327, Y 45.9200, Z -3.8333, A 0.000, B 0.000, C 0.000 }
gfCNCPoint2[28312] = {X 277.3960, Y 45.9200, Z -3.8333, A 0.000, B 0.000, C 0.000 }
gfCNCPoint2[28313] = {X 277.3539, Y 45.4857, Z -3.8333, A 0.000, B 0.000, C 0.000 }
gfCNCPoint2[28314] = {X 277.3378, Y 45.0497, Z -3.8333, A 0.000, B 0.000, C 0.000 }
gfCNCPoint2[28315] = {X 277.3377, Y 44.1979, Z -3.8333, A 0.000, B 0.000, C 0.000 }
gfCNCPoint2[28316] = {X 277.4031, Y 43.2532, Z -3.8333, A 0.000, B 0.000, C 0.000 }
gfCNCPoint2[28317] = {X 277.5897, Y 42.3249, Z -3.8333, A 0.000, B 0.000, C 0.000 }
gfCNCPoint2[28318] = {X 277.8945, Y 41.4283, Z -3.8333, A 0.000, B 0.000, C 0.000 }
gfCNCPoint2[28319] = {X 278.3244, Y 40.5575, Z -3.8333, A 0.000, B 0.000, C 0.000 }
gfCNCPoint2[28320] = {X 278.8656, Y 39.7512, Z -3.8333, A 0.000, B 0.000, C 0.000 }
gfCNCPoint2[28321] = {X 278.8652, Y 17.4398, Z -3.8333, A 0.000, B 0.000, C 0.000 }
gfCNCPoint2[28322] = {X 278.3224, Y 16.6343, Z -3.8333, A 0.000, B 0.000, C 0.000 }
gfCNCPoint2[28323] = {X 277.8917, Y 15.7637, Z -3.8333, A 0.000, B 0.000, C 0.000 }
gfCNCPoint2[28324] = {X 277.5902, Y 14.8788, Z -3.8333, A 0.000, B 0.000, C 0.000 }
gfCNCPoint2[28325] = {X 277.4046, Y 13.9627, Z -3.8333, A 0.000, B 0.000, C 0.000 }
gfCNCPoint2[28326] = {X 277.3379, Y 13.0303, Z -3.8333, A 0.000, B 0.000, C 0.000 }
gfCNCPoint2[28327] = {X 277.3377, Y 12.1868, Z -3.8333, A 0.000, B 0.000, C 0.000 }
gfCNCPoint2[28328] = {X 277.3952, Y 11.2737, Z -3.8333, A 0.000, B 0.000, C 0.000 }
gfCNCPoint2[28329] = {X 277.5667, Y 10.3751, Z -3.8333, A 0.000, B 0.000, C 0.000 }
gfCNCPoint2[28330] = {X 277.8496, Y 9.5050, Z -3.8333, A 0.000, B 0.000, C 0.000 }
gfCNCPoint2[28331] = {X 273.4967, Y 9.5050, Z -3.8333, A 0.000, B 0.000, C 0.000 }
gfCNCPoint2[28332] = {X 273.7799, Y 10.3733, Z -3.8333, A 0.000, B 0.000, C 0.000 }
gfCNCPoint2[28333] = {X 273.9523, Y 11.2701, Z -3.8333, A 0.000, B 0.000, C 0.000 }
gfCNCPoint2[28334] = {X 274.0110, Y 12.1816, Z -3.8333, A 0.000, B 0.000, C 0.000 }
gfCNCPoint2[28335] = {X 274.0107, Y 13.0462, Z -3.8333, A 0.000, B 0.000, C 0.000 }
gfCNCPoint2[28336] = {X 273.9427, Y 13.9732, Z -3.8333, A 0.000, B 0.000, C 0.000 }
gfCNCPoint2[28337] = {X 273.7571, Y 14.8840, Z -3.8333, A 0.000, B 0.000, C 0.000 }
gfCNCPoint2[28338] = {X 273.4570, Y 15.7637, Z -3.8333, A 0.000, B 0.000, C 0.000 }
gfCNCPoint2[28339] = {X 271.2396, Y 14.8453, Z -3.8333, A 0.000, B 0.000, C 0.000 }
gfCNCPoint2[28340] = {X 270.7503, Y 15.7457, Z -3.8333, A 0.000, B 0.000, C 0.000 }
gfCNCPoint2[28341] = {X 270.0837, Y 16.5240, Z -3.8333, A 0.000, B 0.000, C 0.000 }
gfCNCPoint2[28342] = {X 270.0836, Y 40.6627, Z -3.8333, A 0.000, B 0.000, C 0.000 }
gfCNCPoint2[28343] = {X 270.7241, Y 41.4035, Z -3.8333, A 0.000, B 0.000, C 0.000 }
gfCNCPoint2[28344] = {X 271.2039, Y 42.2574, Z -3.8333, A 0.000, B 0.000, C 0.000 }
gfCNCPoint2[28345] = {X 271.5035, Y 43.1898, Z -3.8333, A 0.000, B 0.000, C 0.000 }
gfCNCPoint2[28346] = {X 271.6108, Y 44.1633, Z -3.8333, A 0.000, B 0.000, C 0.000 }
gfCNCPoint2[28347] = {X 271.6110, Y 45.0000, Z -3.8333, A 0.000, B 0.000, C 0.000 }
gfCNCPoint2[28348] = {X 271.5959, Y 45.3844, Z -3.8333, A 0.000, B 0.000, C 0.000 }
gfCNCPoint2[28349] = {X 271.5505, Y 45.7664, Z -3.8333, A 0.000, B 0.000, C 0.000 }
gfCNCPoint2[28350] = {X 271.2989, Y 46.7171, Z -3.8333, A 0.000, B 0.000, C 0.000 }
gfCNCPoint2[28351] = {X 270.8619, Y 47.5982, Z -3.8333, A 0.000, B 0.000, C 0.000 }
gfCNCPoint2[28352] = {X 270.2571, Y 48.3736, Z -3.8333, A 0.000, B 0.000, C 0.000 }
gfCNCPoint2[28353] = {X 269.5090, Y 49.0121, Z -3.8333, A 0.000, B 0.000, C 0.000 }
gfCNCPoint2[28354] = {X 268.6482, Y 49.4876, Z -3.8333, A 0.000, B 0.000, C 0.000 }
gfCNCPoint2[28355] = {X 267.7095, Y 49.7809, Z -3.8333, A 0.000, B 0.000, C 0.000 }
gfCNCPoint2[28356] = {X 266.7310, Y 49.8800, Z -3.8333, A 0.000, B 0.000, C 0.000 }
gfCNCPoint2[28357] = {X 260.2876, Y 49.8800, Z -3.8333, A 0.000, B 0.000, C 0.000 }
gfCNCPoint2[28358] = {X 259.2646, Y 49.7716, Z -3.8333, A 0.000, B 0.000, C 0.000 }
gfCNCPoint2[28359] = {X 258.2870, Y 49.4511, Z -3.8333, A 0.000, B 0.000, C 0.000 }
gfCNCPoint2[28360] = {X 257.3984, Y 48.9328, Z -3.8333, A 0.000, B 0.000, C 0.000 }
gfCNCPoint2[28361] = {X 256.6382, Y 48.2398, Z -3.8333, A 0.000, B 0.000, C 0.000 }
gfCNCPoint2[28362] = {X 256.0401, Y 47.4028, Z -3.8333, A 0.000, B 0.000, C 0.000 }
gfCNCPoint2[28363] = {X 255.6308, Y 46.4590, Z -3.8333, A 0.000, B 0.000, C 0.000 }
gfCNCPoint2[28364] = {X 255.4666, Y 45.7568, Z -3.8333, A 0.000, B 0.000, C 0.000 }
gfCNCPoint2[28365] = {X 255.4077, Y 45.0380, Z -3.8333, A 0.000, B 0.000, C 0.000 }
gfCNCPoint2[28366] = {X 255.4080, Y 44.1417, Z -3.8333, A 0.000, B 0.000, C 0.000 }
gfCNCPoint2[28367] = {X 255.5183, Y 43.1751, Z -3.8333, A 0.000, B 0.000, C 0.000 }
gfCNCPoint2[28368] = {X 255.8181, Y 42.2497, Z -3.8333, A 0.000, B 0.000, C 0.000 }
gfCNCPoint2[28369] = {X 256.2955, Y 41.4021, Z -3.8333, A 0.000, B 0.000, C 0.000 }
gfCNCPoint2[28370] = {X 256.9315, Y 40.6660, Z -3.8333, A 0.000, B 0.000, C 0.000 }
gfCNCPoint2[28371] = {X 256.9315, Y 35.0338, Z -3.8333, A 0.000, B 0.000, C 0.000 }
gfCNCPoint2[28372] = {X 255.1094, Y 35.0338, Z -3.8333, A 0.000, B 0.000, C 0.000 }
gfCNCPoint2[28373] = {X 251.0865, Y 42.8705, Z -3.8333, A 0.000, B 0.000, C 0.000 }
gfCNCPoint2[28374] = {X 251.2237, Y 43.5127, Z -3.8333, A 0.000, B 0.000, C 0.000 }
gfCNCPoint2[28375] = {X 251.2734, Y 44.1675, Z -3.8333, A 0.000, B 0.000, C 0.000 }
gfCNCPoint2[28376] = {X 251.2736, Y 45.0000, Z -3.8333, A 0.000, B 0.000, C 0.000 }
gfCNCPoint2[28377] = {X 251.2174, Y 45.7380, Z -3.8333, A 0.000, B 0.000, C 0.000 }
gfCNCPoint2[28378] = {X 251.0503, Y 46.4590, Z -3.8333, A 0.000, B 0.000, C 0.000 }
gfCNCPoint2[28379] = {X 250.6346, Y 47.4142, Z -3.8333, A 0.000, B 0.000, C 0.000 }
gfCNCPoint2[28380] = {X 250.0255, Y 48.2593, Z -3.8333, A 0.000, B 0.000, C 0.000 }
gfCNCPoint2[28381] = {X 249.2510, Y 48.9560, Z -3.8333, A 0.000, B 0.000, C 0.000 }
gfCNCPoint2[28382] = {X 248.3462, Y 49.4723, Z -3.8333, A 0.000, B 0.000, C 0.000 }
gfCNCPoint2[28383] = {X 247.3525, Y 49.7849, Z -3.8333, A 0.000, B 0.000, C 0.000 }
gfCNCPoint2[28384] = {X 246.8754, Y 49.8562, Z -3.8333, A 0.000, B 0.000, C 0.000 }
gfCNCPoint2[28385] = {X 246.3936, Y 49.8800, Z -3.8333, A 0.000, B 0.000, C 0.000 }
gfCNCPoint2[28386] = {X 242.5312, Y 49.8800, Z -3.8333, A 0.000, B 0.000, C 0.000 }
gfCNCPoint2[28387] = {X 242.5312, Y 49.4000, Z -3.8333, A 0.000, B 0.000, C 0.000 }
gfCNCPoint2[28388] = {X 239.8075, Y 49.4000, Z -3.8333, A 0.000, B 0.000, C 0.000 }
gfCNCPoint2[28389] = {X 238.8284, Y 49.2897, Z -3.8333, A 0.000, B 0.000, C 0.000 }
gfCNCPoint2[28390] = {X 237.8984, Y 48.9643, Z -3.8333, A 0.000, B 0.000, C 0.000 }
gfCNCPoint2[28391] = {X 237.0641, Y 48.4401, Z -3.8333, A 0.000, B 0.000, C 0.000 }
gfCNCPoint2[28392] = {X 236.3674, Y 47.7434, Z -3.8333, A 0.000, B 0.000, C 0.000 }
gfCNCPoint2[28393] = {X 235.8432, Y 46.9091, Z -3.8333, A 0.000, B 0.000, C 0.000 }
gfCNCPoint2[28394] = {X 235.5178, Y 45.9791, Z -3.8333, A 0.000, B 0.000, C 0.000 }
gfCNCPoint2[28395] = {X 235.4075, Y 45.0000, Z -3.8333, A 0.000, B 0.000, C 0.000 }
gfCNCPoint2[28396] = {X 235.4079, Y 44.1483, Z -3.8333, A 0.000, B 0.000, C 0.000 }
gfCNCPoint2[28397] = {X 235.5063, Y 43.2816, Z -3.8333, A 0.000, B 0.000, C 0.000 }
gfCNCPoint2[28398] = {X 235.7737, Y 42.4514, Z -3.8333, A 0.000, B 0.000, C 0.000 }
gfCNCPoint2[28399] = {X 236.1996, Y 41.6903, Z -3.8333, A 0.000, B 0.000, C 0.000 }
gfCNCPoint2[28400] = {X 236.7672, Y 41.0281, Z -3.8333, A 0.000, B 0.000, C 0.000 }
gfCNCPoint2[28401] = {X 237.4544, Y 40.4909, Z -3.8333, A 0.000, B 0.000, C 0.000 }
gfCNCPoint2[28402] = {X 238.2339, Y 40.0998, Z -3.8333, A 0.000, B 0.000, C 0.000 }
gfCNCPoint2[28403] = {X 242.1749, Y 32.3858, Z -3.8333, A 0.000, B 0.000, C 0.000 }
gfCNCPoint2[28404] = {X 241.0114, Y 31.5934, Z -3.8333, A 0.000, B 0.000, C 0.000 }
gfCNCPoint2[28405] = {X 239.9544, Y 30.6637, Z -3.8333, A 0.000, B 0.000, C 0.000 }
gfCNCPoint2[28406] = {X 239.0201, Y 29.6107, Z -3.8333, A 0.000, B 0.000, C 0.000 }
gfCNCPoint2[28407] = {X 238.2227, Y 28.4505, Z -3.8333, A 0.000, B 0.000, C 0.000 }
gfCNCPoint2[28408] = {X 237.5745, Y 27.2009, Z -3.8333, A 0.000, B 0.000, C 0.000 }
gfCNCPoint2[28409] = {X 237.0853, Y 25.8809, Z -3.8333, A 0.000, B 0.000, C 0.000 }
gfCNCPoint2[28410] = {X 236.6635, Y 24.0613, Z -3.8333, A 0.000, B 0.000, C 0.000 }
gfCNCPoint2[28411] = {X 236.4487, Y 22.2057, Z -3.8333, A 0.000, B 0.000, C 0.000 }
gfCNCPoint2[28412] = {X 236.4435, Y 20.3378, Z -3.8333, A 0.000, B 0.000, C 0.000 }
gfCNCPoint2[28413] = {X 236.6479, Y 18.4811, Z -3.8333, A 0.000, B 0.000, C 0.000 }
gfCNCPoint2[28414] = {X 237.0595, Y 16.6591, Z -3.8333, A 0.000, B 0.000, C 0.000 }
gfCNCPoint2[28415] = {X 237.6337, Y 15.0729, Z -3.8333, A 0.000, B 0.000, C 0.000 }
gfCNCPoint2[28416] = {X 238.4260, Y 13.5835, Z -3.8333, A 0.000, B 0.000, C 0.000 }
gfCNCPoint2[28417] = {X 239.4204, Y 12.2208, Z -3.8333, A 0.000, B 0.000, C 0.000 }
gfCNCPoint2[28418] = {X 240.5971, Y 11.0121, Z -3.8333, A 0.000, B 0.000, C 0.000 }
gfCNCPoint2[28419] = {X 241.9326, Y 9.9814, Z -3.8333, A 0.000, B 0.000, C 0.000 }
gfCNCPoint2[28420] = {X 243.4001, Y 9.1495, Z -3.8333, A 0.000, B 0.000, C 0.000 }
gfCNCPoint2[28421] = {X 244.9704, Y 8.5329, Z -3.8333, A 0.000, B 0.000, C 0.000 }
gfCNCPoint2[28422] = {X 246.6119, Y 8.1440, Z -3.8333, A 0.000, B 0.000, C 0.000 }
gfCNCPoint2[28423] = {X 248.7155, Y 7.8717, Z -3.8333, A 0.000, B 0.000, C 0.000 }
gfCNCPoint2[28424] = {X 250.8351, Y 7.7909, Z -3.8333, A 0.000, B 0.000, C 0.000 }
gfCNCPoint2[28425] = {X 266.7640, Y 7.7909, Z -3.8333, A 0.000, B 0.000, C 0.000 }
gfCNCPoint2[28426] = {X 267.7368, Y 7.9078, Z -3.8333, A 0.000, B 0.000, C 0.000 }
gfCNCPoint2[28427] = {X 268.6597, Y 8.2370, Z -3.8333, A 0.000, B 0.000, C 0.000 }
gfCNCPoint2[28428] = {X 269.4869, Y 8.7621, Z -3.8333, A 0.000, B 0.000, C 0.000 }
gfCNCPoint2[28429] = {X 270.1775, Y 9.4571, Z -3.8333, A 0.000, B 0.000, C 0.000 }
gfCNCPoint2[28430] = {X 270.6972, Y 10.2877, Z -3.8333, A 0.000, B 0.000, C 0.000 }
gfCNCPoint2[28431] = {X 271.0204, Y 11.2127, Z -3.8333, A 0.000, B 0.000, C 0.000 }
gfCNCPoint2[28432] = {X 271.1310, Y 12.1862, Z -3.8333, A 0.000, B 0.000, C 0.000 }
gfCNCPoint2[28433] = {X 271.1308, Y 13.0233, Z -3.8333, A 0.000, B 0.000, C 0.000 }
gfCNCPoint2[28434] = {X 271.0225, Y 13.9493, Z -3.8333, A 0.000, B 0.000, C 0.000 }
gfCNCPoint2[28435] = {X 270.7215, Y 14.8316, Z -3.8333, A 0.000, B 0.000, C 0.000 }
gfCNCPoint2[28436] = {X 270.2414, Y 15.6308, Z -3.8333, A 0.000, B 0.000, C 0.000 }
gfCNCPoint2[28437] = {X 269.6037, Y 16.3108, Z -3.8333, A 0.000, B 0.000, C 0.000 }
gfCNCPoint2[28438] = {X 269.6035, Y 40.8758, Z -3.8333, A 0.000, B 0.000, C 0.000 }
gfCNCPoint2[28439] = {X 270.2482, Y 41.5650, Z -3.8333, A 0.000, B 0.000, C 0.000 }
gfCNCPoint2[28440] = {X 270.7310, Y 42.3757, Z -3.8333, A 0.000, B 0.000, C 0.000 }
gfCNCPoint2[28441] = {X 271.0299, Y 43.2707, Z -3.8333, A 0.000, B 0.000, C 0.000 }
gfCNCPoint2[28442] = {X 271.1310, Y 44.2089, Z -3.8333, A 0.000, B 0.000, C 0.000 }
gfCNCPoint2[28443] = {X 271.1310, Y 45.0000, Z -3.8333, A 0.000, B 0.000, C 0.000 }
gfCNCPoint2[28444] = {X 271.0207, Y 45.9791, Z -3.8333, A 0.000, B 0.000, C 0.000 }
gfCNCPoint2[28445] = {X 270.6953, Y 46.9091, Z -3.8333, A 0.000, B 0.000, C 0.000 }
gfCNCPoint2[28446] = {X 270.1711, Y 47.7434, Z -3.8333, A 0.000, B 0.000, C 0.000 }
gfCNCPoint2[28447] = {X 269.4744, Y 48.4401, Z -3.8333, A 0.000, B 0.000, C 0.000 }
gfCNCPoint2[28448] = {X 268.6401, Y 48.9643, Z -3.8333, A 0.000, B 0.000, C 0.000 }
gfCNCPoint2[28449] = {X 267.7101, Y 49.2897, Z -3.8333, A 0.000, B 0.000, C 0.000 }
gfCNCPoint2[28450] = {X 266.7310, Y 49.4000, Z -3.8333, A 0.000, B 0.000, C 0.000 }
gfCNCPoint2[28451] = {X 260.2876, Y 49.4000, Z -3.8333, A 0.000, B 0.000, C 0.000 }
gfCNCPoint2[28452] = {X 259.3085, Y 49.2897, Z -3.8333, A 0.000, B 0.000, C 0.000 }
gfCNCPoint2[28453] = {X 258.3785, Y 48.9643, Z -3.8333, A 0.000, B 0.000, C 0.000 }
gfCNCPoint2[28454] = {X 257.5442, Y 48.4400, Z -3.8333, A 0.000, B 0.000, C 0.000 }
gfCNCPoint2[28455] = {X 256.8475, Y 47.7433, Z -3.8333, A 0.000, B 0.000, C 0.000 }
gfCNCPoint2[28456] = {X 256.3233, Y 46.9091, Z -3.8333, A 0.000, B 0.000, C 0.000 }
gfCNCPoint2[28457] = {X 255.9979, Y 45.9791, Z -3.8333, A 0.000, B 0.000, C 0.000 }
gfCNCPoint2[28458] = {X 255.8876, Y 45.0000, Z -3.8333, A 0.000, B 0.000, C 0.000 }
gfCNCPoint2[28459] = {X 255.8880, Y 44.1483, Z -3.8333, A 0.000, B 0.000, C 0.000 }
gfCNCPoint2[28460] = {X 255.9984, Y 43.2275, Z -3.8333, A 0.000, B 0.000, C 0.000 }
gfCNCPoint2[28461] = {X 256.2993, Y 42.3503, Z -3.8333, A 0.000, B 0.000, C 0.000 }
gfCNCPoint2[28462] = {X 256.7775, Y 41.5556, Z -3.8333, A 0.000, B 0.000, C 0.000 }
gfCNCPoint2[28463] = {X 257.4115, Y 40.8789, Z -3.8333, A 0.000, B 0.000, C 0.000 }
gfCNCPoint2[28464] = {X 257.4115, Y 34.5538, Z -3.8333, A 0.000, B 0.000, C 0.000 }
gfCNCPoint2[28465] = {X 254.8162, Y 34.5538, Z -3.8333, A 0.000, B 0.000, C 0.000 }
gfCNCPoint2[28466] = {X 250.5703, Y 42.8250, Z -3.8333, A 0.000, B 0.000, C 0.000 }
gfCNCPoint2[28467] = {X 250.7374, Y 43.5080, Z -3.8333, A 0.000, B 0.000, C 0.000 }
gfCNCPoint2[28468] = {X 250.7936, Y 44.2089, Z -3.8333, A 0.000, B 0.000, C 0.000 }
gfCNCPoint2[28469] = {X 250.7936, Y 45.0000, Z -3.8333, A 0.000, B 0.000, C 0.000 }
gfCNCPoint2[28470] = {X 250.6832, Y 45.9791, Z -3.8333, A 0.000, B 0.000, C 0.000 }
gfCNCPoint2[28471] = {X 250.3578, Y 46.9091, Z -3.8333, A 0.000, B 0.000, C 0.000 }
gfCNCPoint2[28472] = {X 249.8336, Y 47.7434, Z -3.8333, A 0.000, B 0.000, C 0.000 }
gfCNCPoint2[28473] = {X 249.1369, Y 48.4401, Z -3.8333, A 0.000, B 0.000, C 0.000 }
gfCNCPoint2[28474] = {X 248.3026, Y 48.9643, Z -3.8333, A 0.000, B 0.000, C 0.000 }
gfCNCPoint2[28475] = {X 247.3727, Y 49.2897, Z -3.8333, A 0.000, B 0.000, C 0.000 }
gfCNCPoint2[28476] = {X 246.3936, Y 49.4000, Z -3.8333, A 0.000, B 0.000, C 0.000 }
gfCNCPoint2[28477] = {X 242.5312, Y 49.4000, Z -3.8333, A 0.000, B 0.000, C 0.000 }
gfCNCPoint2[28478] = {X 242.5312, Y 49.8800, Z -3.8333, A 0.000, B 0.000, C 0.000 }
gfCNCPoint2[28479] = {X 243.4812, Y 50.5824, Z -3.8333, A 0.000, B 0.000, C 0.000 }
gfCNCPoint2[28480] = {X 244.3384, Y 51.3953, Z -3.8333, A 0.000, B 0.000, C 0.000 }
gfCNCPoint2[28481] = {X 245.0903, Y 52.3066, Z -3.8333, A 0.000, B 0.000, C 0.000 }
gfCNCPoint2[28482] = {X 245.7256, Y 53.3027, Z -3.8333, A 0.000, B 0.000, C 0.000 }
gfCNCPoint2[28483] = {X 245.9755, Y 53.7843, Z -3.8333, A 0.000, B 0.000, C 0.000 }
gfCNCPoint2[28484] = {X 246.1980, Y 54.2791, Z -3.8333, A 0.000, B 0.000, C 0.000 }
gfCNCPoint2[28485] = {X 249.4596, Y 55.5506, Z -3.8333, A 0.000, B 0.000, C 0.000 }
gfCNCPoint2[28486] = {X 251.8858, Y 56.5133, Z -3.8333, A 0.000, B 0.000, C 0.000 }
gfCNCPoint2[28487] = {X 253.6561, Y 52.0517, Z -3.8333, A 0.000, B 0.000, C 0.000 }
gfCNCPoint2[28488] = {X 253.4966, Y 51.8982, Z -3.8333, A 0.000, B 0.000, C 0.000 }
gfCNCPoint2[28489] = {X 253.3406, Y 51.7410, Z -3.8333, A 0.000, B 0.000, C 0.000 }
gfCNCPoint2[28490] = {X 253.2750, Y 51.8079, Z -3.8333, A 0.000, B 0.000, C 0.000 }
gfCNCPoint2[28491] = {X 253.2088, Y 51.8742, Z -3.8333, A 0.000, B 0.000, C 0.000 }
gfCNCPoint2[28492] = {X 253.6561, Y 52.0517, Z -3.8333, A 0.000, B 0.000, C 0.000 }
gfCNCPoint2[28493] = {X 252.7709, Y 54.2825, Z -3.8333, A 0.000, B 0.000, C 0.000 }
gfCNCPoint2[28494] = {X 259.3950, Y 56.9108, Z -3.8333, A 0.000, B 0.000, C 0.000 }
gfCNCPoint2[28495] = {X 260.2801, Y 54.6800, Z -3.8333, A 0.000, B 0.000, C 0.000 }
gfCNCPoint2[28496] = {X 261.9953, Y 55.3605, Z -3.8333, A 0.000, B 0.000, C 0.000 }
gfCNCPoint2[28497] = {X 262.0628, Y 55.0194, Z -3.8333, A 0.000, B 0.000, C 0.000 }
gfCNCPoint2[28498] = {X 262.1384, Y 54.6800, Z -3.8333, A 0.000, B 0.000, C 0.000 }
gfCNCPoint2[28499] = {X 260.2801, Y 54.6800, Z -3.8333, A 0.000, B 0.000, C 0.000 }
gfCNCPoint2[28500] = {X 259.3950, Y 56.9108, Z -3.8333, A 0.000, B 0.000, C 0.000 }
gfCNCPoint2[28501] = {X 264.1528, Y 58.7987, Z -3.8333, A 0.000, B 0.000, C 0.000 }
gfCNCPoint2[28502] = {X 264.1527, Y 58.0000, Z -3.8333, A 0.000, B 0.000, C 0.000 }
gfCNCPoint2[28503] = {X 264.2034, Y 56.8944, Z -3.8333, A 0.000, B 0.000, C 0.000 }
gfCNCPoint2[28504] = {X 264.3551, Y 55.7980, Z -3.8333, A 0.000, B 0.000, C 0.000 }
gfCNCPoint2[28505] = {X 264.4114, Y 55.5134, Z -3.8333, A 0.000, B 0.000, C 0.000 }
gfCNCPoint2[28506] = {X 264.4745, Y 55.2303, Z -3.8333, A 0.000, B 0.000, C 0.000 }
gfCNCPoint2[28507] = {X 264.9369, Y 53.7185, Z -3.8333, A 0.000, B 0.000, C 0.000 }
gfCNCPoint2[28508] = {X 265.5928, Y 52.2800, Z -3.8333, A 0.000, B 0.000, C 0.000 }
gfCNCPoint2[28509] = {X 260.2876, Y 52.2800, Z -3.8333, A 0.000, B 0.000, C 0.000 }
gfCNCPoint2[28510] = {X 259.1929, Y 52.1972, Z -3.8333, A 0.000, B 0.000, C 0.000 }
gfCNCPoint2[28511] = {X 258.1231, Y 51.9508, Z -3.8333, A 0.000, B 0.000, C 0.000 }
gfCNCPoint2[28512] = {X 257.1025, Y 51.5463, Z -3.8333, A 0.000, B 0.000, C 0.000 }
gfCNCPoint2[28513] = {X 256.1544, Y 50.9929, Z -3.8333, A 0.000, B 0.000, C 0.000 }
gfCNCPoint2[28514] = {X 255.3003, Y 50.3033, Z -3.8333, A 0.000, B 0.000, C 0.000 }
gfCNCPoint2[28515] = {X 255.1803, Y 50.1879, Z -3.8333, A 0.000, B 0.000, C 0.000 }
gfCNCPoint2[28516] = {X 255.0630, Y 50.0697, Z -3.8333, A 0.000, B 0.000, C 0.000 }
gfCNCPoint2[28517] = {X 254.3405, Y 49.1989, Z -3.8333, A 0.000, B 0.000, C 0.000 }
gfCNCPoint2[28518] = {X 253.7617, Y 48.2267, Z -3.8333, A 0.000, B 0.000, C 0.000 }
gfCNCPoint2[28519] = {X 253.3406, Y 47.1766, Z -3.8333, A 0.000, B 0.000, C 0.000 }
gfCNCPoint2[28520] = {X 252.9194, Y 48.2267, Z -3.8333, A 0.000, B 0.000, C 0.000 }
gfCNCPoint2[28521] = {X 252.3406, Y 49.1989, Z -3.8333, A 0.000, B 0.000, C 0.000 }
gfCNCPoint2[28522] = {X 251.6182, Y 50.0697, Z -3.8333, A 0.000, B 0.000, C 0.000 }
gfCNCPoint2[28523] = {X 251.5689, Y 50.1200, Z -3.8333, A 0.000, B 0.000, C 0.000 }
gfCNCPoint2[28524] = {X 251.5191, Y 50.1698, Z -3.8333, A 0.000, B 0.000, C 0.000 }
gfCNCPoint2[28525] = {X 250.7135, Y 50.8598, Z -3.8333, A 0.000, B 0.000, C 0.000 }
gfCNCPoint2[28526] = {X 249.8161, Y 51.4253, Z -3.8333, A 0.000, B 0.000, C 0.000 }
gfCNCPoint2[28527] = {X 248.8461, Y 51.8544, Z -3.8333, A 0.000, B 0.000, C 0.000 }
gfCNCPoint2[28528] = {X 247.8241, Y 52.1381, Z -3.8333, A 0.000, B 0.000, C 0.000 }
gfCNCPoint2[28529] = {X 247.8928, Y 52.2637, Z -3.8333, A 0.000, B 0.000, C 0.000 }
gfCNCPoint2[28530] = {X 247.9601, Y 52.3901, Z -3.8333, A 0.000, B 0.000, C 0.000 }
gfCNCPoint2[28531] = {X 250.3415, Y 53.3185, Z -3.8333, A 0.000, B 0.000, C 0.000 }
gfCNCPoint2[28532] = {X 252.7709, Y 54.2825, Z -3.8333, A 0.000, B 0.000, C 0.000 }
gfCNCPoint2[28533] = {X 251.8858, Y 56.5133, Z -3.8333, A 0.000, B 0.000, C 0.000 }
gfCNCPoint2[28534] = {X 267.2830, Y 62.6227, Z -3.8333, A 0.000, B 0.000, C 0.000 }
gfCNCPoint2[28535] = {X 266.8847, Y 61.4474, Z -3.8333, A 0.000, B 0.000, C 0.000 }
gfCNCPoint2[28536] = {X 266.6399, Y 60.2309, Z -3.8333, A 0.000, B 0.000, C 0.000 }
gfCNCPoint2[28537] = {X 266.5529, Y 58.9930, Z -3.8333, A 0.000, B 0.000, C 0.000 }
gfCNCPoint2[28538] = {X 266.5527, Y 58.0000, Z -3.8333, A 0.000, B 0.000, C 0.000 }
gfCNCPoint2[28539] = {X 266.6262, Y 56.8093, Z -3.8333, A 0.000, B 0.000, C 0.000 }
gfCNCPoint2[28540] = {X 266.8456, Y 55.6367, Z -3.8333, A 0.000, B 0.000, C 0.000 }
gfCNCPoint2[28541] = {X 267.2076, Y 54.5000, Z -3.8333, A 0.000, B 0.000, C 0.000 }
gfCNCPoint2[28542] = {X 267.7067, Y 53.4164, Z -3.8333, A 0.000, B 0.000, C 0.000 }
gfCNCPoint2[28543] = {X 268.4728, Y 52.2132, Z -3.8333, A 0.000, B 0.000, C 0.000 }
gfCNCPoint2[28544] = {X 269.4075, Y 51.1357, Z -3.8333, A 0.000, B 0.000, C 0.000 }
gfCNCPoint2[28545] = {X 270.4903, Y 50.2072, Z -3.8333, A 0.000, B 0.000, C 0.000 }
gfCNCPoint2[28546] = {X 271.6979, Y 49.4479, Z -3.8333, A 0.000, B 0.000, C 0.000 }
gfCNCPoint2[28547] = {X 273.0039, Y 48.8744, Z -3.8333, A 0.000, B 0.000, C 0.000 }
gfCNCPoint2[28548] = {X 274.3800, Y 48.4989, Z -3.8333, A 0.000, B 0.000, C 0.000 }
gfCNCPoint2[28549] = {X 275.3020, Y 48.3648, Z -3.8333, A 0.000, B 0.000, C 0.000 }
gfCNCPoint2[28550] = {X 276.2327, Y 48.3200, Z -3.8333, A 0.000, B 0.000, C 0.000 }
gfCNCPoint2[28551] = {X 281.0411, Y 48.3200, Z -3.8333, A 0.000, B 0.000, C 0.000 }
gfCNCPoint2[28552] = {X 280.4347, Y 47.5134, Z -3.8333, A 0.000, B 0.000, C 0.000 }
gfCNCPoint2[28553] = {X 280.0072, Y 46.5992, Z -3.8333, A 0.000, B 0.000, C 0.000 }
gfCNCPoint2[28554] = {X 279.7768, Y 45.6167, Z -3.8333, A 0.000, B 0.000, C 0.000 }
gfCNCPoint2[28555] = {X 279.7488, Y 45.3288, Z -3.8333, A 0.000, B 0.000, C 0.000 }
gfCNCPoint2[28556] = {X 279.7378, Y 45.0398, Z -3.8333, A 0.000, B 0.000, C 0.000 }
gfCNCPoint2[28557] = {X 279.7377, Y 44.2042, Z -3.8333, A 0.000, B 0.000, C 0.000 }
gfCNCPoint2[28558] = {X 279.8422, Y 43.2206, Z -3.8333, A 0.000, B 0.000, C 0.000 }
gfCNCPoint2[28559] = {X 280.1409, Y 42.2777, Z -3.8333, A 0.000, B 0.000, C 0.000 }
gfCNCPoint2[28560] = {X 280.6219, Y 41.4135, Z -3.8333, A 0.000, B 0.000, C 0.000 }
gfCNCPoint2[28561] = {X 281.2656, Y 40.6626, Z -3.8333, A 0.000, B 0.000, C 0.000 }
gfCNCPoint2[28562] = {X 281.2652, Y 16.5242, Z -3.8333, A 0.000, B 0.000, C 0.000 }
gfCNCPoint2[28563] = {X 280.6241, Y 15.7826, Z -3.8333, A 0.000, B 0.000, C 0.000 }
gfCNCPoint2[28564] = {X 280.1441, Y 14.9278, Z -3.8333, A 0.000, B 0.000, C 0.000 }
gfCNCPoint2[28565] = {X 279.8447, Y 13.9943, Z -3.8333, A 0.000, B 0.000, C 0.000 }
gfCNCPoint2[28566] = {X 279.7378, Y 13.0198, Z -3.8333, A 0.000, B 0.000, C 0.000 }
gfCNCPoint2[28567] = {X 279.7377, Y 12.1868, Z -3.8333, A 0.000, B 0.000, C 0.000 }
gfCNCPoint2[28568] = {X 279.8242, Y 11.2717, Z -3.8333, A 0.000, B 0.000, C 0.000 }
gfCNCPoint2[28569] = {X 280.0809, Y 10.3891, Z -3.8333, A 0.000, B 0.000, C 0.000 }
gfCNCPoint2[28570] = {X 280.5256, Y 9.5280, Z -3.8333, A 0.000, B 0.000, C 0.000 }
gfCNCPoint2[28571] = {X 281.1317, Y 8.7718, Z -3.8333, A 0.000, B 0.000, C 0.000 }
gfCNCPoint2[28572] = {X 281.8753, Y 8.1503, Z -3.8333, A 0.000, B 0.000, C 0.000 }
gfCNCPoint2[28573] = {X 282.7270, Y 7.6879, Z -3.8333, A 0.000, B 0.000, C 0.000 }
gfCNCPoint2[28574] = {X 283.6533, Y 7.4030, Z -3.8333, A 0.000, B 0.000, C 0.000 }
gfCNCPoint2[28575] = {X 284.6177, Y 7.3068, Z -3.8333, A 0.000, B 0.000, C 0.000 }
gfCNCPoint2[28576] = {X 291.0611, Y 7.3068, Z -3.8333, A 0.000, B 0.000, C 0.000 }
gfCNCPoint2[28577] = {X 292.0255, Y 7.4030, Z -3.8333, A 0.000, B 0.000, C 0.000 }
gfCNCPoint2[28578] = {X 292.9518, Y 7.6879, Z -3.8333, A 0.000, B 0.000, C 0.000 }
gfCNCPoint2[28579] = {X 293.8035, Y 8.1503, Z -3.8333, A 0.000, B 0.000, C 0.000 }
gfCNCPoint2[28580] = {X 294.5471, Y 8.7718, Z -3.8333, A 0.000, B 0.000, C 0.000 }
gfCNCPoint2[28581] = {X 295.1532, Y 9.5280, Z -3.8333, A 0.000, B 0.000, C 0.000 }
gfCNCPoint2[28582] = {X 295.5980, Y 10.3891, Z -3.8333, A 0.000, B 0.000, C 0.000 }
gfCNCPoint2[28583] = {X 295.8044, Y 11.0397, Z -3.8333, A 0.000, B 0.000, C 0.000 }
gfCNCPoint2[28584] = {X 295.9181, Y 11.7127, Z -3.8333, A 0.000, B 0.000, C 0.000 }
gfCNCPoint2[28585] = {X 295.9354, Y 11.9495, Z -3.8333, A 0.000, B 0.000, C 0.000 }
gfCNCPoint2[28586] = {X 295.9411, Y 12.1868, Z -3.8333, A 0.000, B 0.000, C 0.000 }
gfCNCPoint2[28587] = {X 295.9409, Y 13.0237, Z -3.8333, A 0.000, B 0.000, C 0.000 }
gfCNCPoint2[28588] = {X 295.9342, Y 13.2382, Z -3.8333, A 0.000, B 0.000, C 0.000 }
gfCNCPoint2[28589] = {X 295.9180, Y 13.4521, Z -3.8333, A 0.000, B 0.000, C 0.000 }
gfCNCPoint2[28590] = {X 298.3067, Y 13.6853, Z -3.8333, A 0.000, B 0.000, C 0.000 }
gfCNCPoint2[28591] = {X 298.1361, Y 14.6937, Z -3.8333, A 0.000, B 0.000, C 0.000 }
gfCNCPoint2[28592] = {X 297.8258, Y 15.6683, Z -3.8333, A 0.000, B 0.000, C 0.000 }
gfCNCPoint2[28593] = {X 297.3820, Y 16.5897, Z -3.8333, A 0.000, B 0.000, C 0.000 }
gfCNCPoint2[28594] = {X 296.8135, Y 17.4399, Z -3.8333, A 0.000, B 0.000, C 0.000 }
gfCNCPoint2[28595] = {X 296.8139, Y 19.2365, Z -3.8333, A 0.000, B 0.000, C 0.000 }
gfCNCPoint2[28596] = {X 299.7995, Y 19.2365, Z -3.8333, A 0.000, B 0.000, C 0.000 }
gfCNCPoint2[28597] = {X 299.7996, Y 17.4396, Z -3.8333, A 0.000, B 0.000, C 0.000 }
gfCNCPoint2[28598] = {X 299.2312, Y 16.5895, Z -3.8333, A 0.000, B 0.000, C 0.000 }
gfCNCPoint2[28599] = {X 298.7875, Y 15.6681, Z -3.8333, A 0.000, B 0.000, C 0.000 }
gfCNCPoint2[28600] = {X 298.4773, Y 14.6936, Z -3.8333, A 0.000, B 0.000, C 0.000 }
gfCNCPoint2[28601] = {X 298.3067, Y 13.6853, Z -3.8333, A 0.000, B 0.000, C 0.000 }
gfCNCPoint2[28602] = {X 295.9180, Y 13.4521, Z -3.8333, A 0.000, B 0.000, C 0.000 }
gfCNCPoint2[28603] = {X 295.7560, Y 14.3096, Z -3.8333, A 0.000, B 0.000, C 0.000 }
gfCNCPoint2[28604] = {X 295.4437, Y 15.1245, Z -3.8333, A 0.000, B 0.000, C 0.000 }
gfCNCPoint2[28605] = {X 294.9914, Y 15.8707, Z -3.8333, A 0.000, B 0.000, C 0.000 }
gfCNCPoint2[28606] = {X 294.4133, Y 16.5245, Z -3.8333, A 0.000, B 0.000, C 0.000 }
gfCNCPoint2[28607] = {X 294.4143, Y 21.6365, Z -3.8333, A 0.000, B 0.000, C 0.000 }
gfCNCPoint2[28608] = {X 302.1993, Y 21.6365, Z -3.8333, A 0.000, B 0.000, C 0.000 }
gfCNCPoint2[28609] = {X 302.1997, Y 16.5241, Z -3.8333, A 0.000, B 0.000, C 0.000 }
gfCNCPoint2[28610] = {X 301.6218, Y 15.8704, Z -3.8333, A 0.000, B 0.000, C 0.000 }
gfCNCPoint2[28611] = {X 301.1695, Y 15.1242, Z -3.8333, A 0.000, B 0.000, C 0.000 }
gfCNCPoint2[28612] = {X 300.8574, Y 14.3095, Z -3.8333, A 0.000, B 0.000, C 0.000 }
gfCNCPoint2[28613] = {X 300.6953, Y 13.4521, Z -3.8333, A 0.000, B 0.000, C 0.000 }
gfCNCPoint2[28614] = {X 300.6791, Y 13.2371, Z -3.8333, A 0.000, B 0.000, C 0.000 }
gfCNCPoint2[28615] = {X 300.6724, Y 13.0215, Z -3.8333, A 0.000, B 0.000, C 0.000 }
gfCNCPoint2[28616] = {X 300.6723, Y 12.1868, Z -3.8333, A 0.000, B 0.000, C 0.000 }
gfCNCPoint2[28617] = {X 300.6780, Y 11.9495, Z -3.8333, A 0.000, B 0.000, C 0.000 }
gfCNCPoint2[28618] = {X 300.6953, Y 11.7127, Z -3.8333, A 0.000, B 0.000, C 0.000 }
gfCNCPoint2[28619] = {X 300.8090, Y 11.0397, Z -3.8333, A 0.000, B 0.000, C 0.000 }
gfCNCPoint2[28620] = {X 301.0154, Y 10.3891, Z -3.8333, A 0.000, B 0.000, C 0.000 }
gfCNCPoint2[28621] = {X 301.4602, Y 9.5280, Z -3.8333, A 0.000, B 0.000, C 0.000 }
gfCNCPoint2[28622] = {X 302.0663, Y 8.7718, Z -3.8333, A 0.000, B 0.000, C 0.000 }
gfCNCPoint2[28623] = {X 302.8098, Y 8.1503, Z -3.8333, A 0.000, B 0.000, C 0.000 }
gfCNCPoint2[28624] = {X 303.6616, Y 7.6879, Z -3.8333, A 0.000, B 0.000, C 0.000 }
gfCNCPoint2[28625] = {X 304.5879, Y 7.4030, Z -3.8333, A 0.000, B 0.000, C 0.000 }
gfCNCPoint2[28626] = {X 305.5523, Y 7.3068, Z -3.8333, A 0.000, B 0.000, C 0.000 }
gfCNCPoint2[28627] = {X 311.9957, Y 7.3068, Z -3.8333, A 0.000, B 0.000, C 0.000 }
gfCNCPoint2[28628] = {X 312.9478, Y 7.4006, Z -3.8333, A 0.000, B 0.000, C 0.000 }
gfCNCPoint2[28629] = {X 313.8632, Y 7.6783, Z -3.8333, A 0.000, B 0.000, C 0.000 }
gfCNCPoint2[28630] = {X 314.7069, Y 8.1292, Z -3.8333, A 0.000, B 0.000, C 0.000 }
gfCNCPoint2[28631] = {X 315.4464, Y 8.7361, Z -3.8333, A 0.000, B 0.000, C 0.000 }
gfCNCPoint2[28632] = {X 316.0533, Y 9.4756, Z -3.8333, A 0.000, B 0.000, C 0.000 }
gfCNCPoint2[28633] = {X 316.5043, Y 10.3193, Z -3.8333, A 0.000, B 0.000, C 0.000 }
gfCNCPoint2[28634] = {X 316.7820, Y 11.2348, Z -3.8333, A 0.000, B 0.000, C 0.000 }
gfCNCPoint2[28635] = {X 316.8757, Y 12.1868, Z -3.8333, A 0.000, B 0.000, C 0.000 }
gfCNCPoint2[28636] = {X 316.8755, Y 13.0237, Z -3.8333, A 0.000, B 0.000, C 0.000 }
gfCNCPoint2[28637] = {X 316.7681, Y 13.9972, Z -3.8333, A 0.000, B 0.000, C 0.000 }
gfCNCPoint2[28638] = {X 316.4685, Y 14.9297, Z -3.8333, A 0.000, B 0.000, C 0.000 }
gfCNCPoint2[28639] = {X 315.9887, Y 15.7835, Z -3.8333, A 0.000, B 0.000, C 0.000 }
gfCNCPoint2[28640] = {X 315.3480, Y 16.5243, Z -3.8333, A 0.000, B 0.000, C 0.000 }
gfCNCPoint2[28641] = {X 315.3478, Y 40.6622, Z -3.8333, A 0.000, B 0.000, C 0.000 }
gfCNCPoint2[28642] = {X 315.9890, Y 41.4038, Z -3.8333, A 0.000, B 0.000, C 0.000 }
gfCNCPoint2[28643] = {X 316.4691, Y 42.2585, Z -3.8333, A 0.000, B 0.000, C 0.000 }
gfCNCPoint2[28644] = {X 316.7686, Y 43.1919, Z -3.8333, A 0.000, B 0.000, C 0.000 }
gfCNCPoint2[28645] = {X 316.8755, Y 44.1664, Z -3.8333, A 0.000, B 0.000, C 0.000 }
gfCNCPoint2[28646] = {X 316.8757, Y 45.0000, Z -3.8333, A 0.000, B 0.000, C 0.000 }
gfCNCPoint2[28647] = {X 316.8749, Y 45.0899, Z -3.8333, A 0.000, B 0.000, C 0.000 }
gfCNCPoint2[28648] = {X 316.8724, Y 45.1799, Z -3.8333, A 0.000, B 0.000, C 0.000 }
gfCNCPoint2[28649] = {X 316.8594, Y 45.3987, Z -3.8333, A 0.000, B 0.000, C 0.000 }
gfCNCPoint2[28650] = {X 316.8366, Y 45.6167, Z -3.8333, A 0.000, B 0.000, C 0.000 }
gfCNCPoint2[28651] = {X 316.6062, Y 46.5992, Z -3.8333, A 0.000, B 0.000, C 0.000 }
gfCNCPoint2[28652] = {X 316.1787, Y 47.5134, Z -3.8333, A 0.000, B 0.000, C 0.000 }
gfCNCPoint2[28653] = {X 315.5723, Y 48.3200, Z -3.8333, A 0.000, B 0.000, C 0.000 }
gfCNCPoint2[28654] = {X 315.2205, Y 47.9934, Z -3.8333, A 0.000, B 0.000, C 0.000 }
gfCNCPoint2[28655] = {X 314.5413, Y 48.5889, Z -3.8333, A 0.000, B 0.000, C 0.000 }
gfCNCPoint2[28656] = {X 313.7548, Y 49.0331, Z -3.8333, A 0.000, B 0.000, C 0.000 }
gfCNCPoint2[28657] = {X 312.8942, Y 49.3073, Z -3.8333, A 0.000, B 0.000, C 0.000 }
gfCNCPoint2[28658] = {X 311.9957, Y 49.4000, Z -3.8333, A 0.000, B 0.000, C 0.000 }
gfCNCPoint2[28659] = {X 305.5523, Y 49.4000, Z -3.8333, A 0.000, B 0.000, C 0.000 }
gfCNCPoint2[28660] = {X 304.5732, Y 49.2897, Z -3.8333, A 0.000, B 0.000, C 0.000 }
gfCNCPoint2[28661] = {X 303.6432, Y 48.9643, Z -3.8333, A 0.000, B 0.000, C 0.000 }
gfCNCPoint2[28662] = {X 302.8089, Y 48.4400, Z -3.8333, A 0.000, B 0.000, C 0.000 }
gfCNCPoint2[28663] = {X 302.1122, Y 47.7433, Z -3.8333, A 0.000, B 0.000, C 0.000 }
gfCNCPoint2[28664] = {X 301.5880, Y 46.9091, Z -3.8333, A 0.000, B 0.000, C 0.000 }
gfCNCPoint2[28665] = {X 301.2626, Y 45.9791, Z -3.8333, A 0.000, B 0.000, C 0.000 }
gfCNCPoint2[28666] = {X 301.1523, Y 45.0000, Z -3.8333, A 0.000, B 0.000, C 0.000 }
gfCNCPoint2[28667] = {X 301.1524, Y 44.1993, Z -3.8333, A 0.000, B 0.000, C 0.000 }
gfCNCPoint2[28668] = {X 301.2702, Y 43.2558, Z -3.8333, A 0.000, B 0.000, C 0.000 }
gfCNCPoint2[28669] = {X 301.5733, Y 42.3547, Z -3.8333, A 0.000, B 0.000, C 0.000 }
gfCNCPoint2[28670] = {X 302.0496, Y 41.5318, Z -3.8333, A 0.000, B 0.000, C 0.000 }
gfCNCPoint2[28671] = {X 302.6801, Y 40.8202, Z -3.8333, A 0.000, B 0.000, C 0.000 }
gfCNCPoint2[28672] = {X 302.6801, Y 34.1143, Z -3.8333, A 0.000, B 0.000, C 0.000 }
gfCNCPoint2[28673] = {X 293.9342, Y 34.1143, Z -3.8333, A 0.000, B 0.000, C 0.000 }
gfCNCPoint2[28674] = {X 293.9334, Y 40.8661, Z -3.8333, A 0.000, B 0.000, C 0.000 }
gfCNCPoint2[28675] = {X 294.5734, Y 41.5611, Z -3.8333, A 0.000, B 0.000, C 0.000 }
gfCNCPoint2[28676] = {X 295.0541, Y 42.3744, Z -3.8333, A 0.000, B 0.000, C 0.000 }
gfCNCPoint2[28677] = {X 295.3545, Y 43.2702, Z -3.8333, A 0.000, B 0.000, C 0.000 }
gfCNCPoint2[28678] = {X 295.4611, Y 44.2089, Z -3.8333, A 0.000, B 0.000, C 0.000 }
gfCNCPoint2[28679] = {X 295.4611, Y 45.0000, Z -3.8333, A 0.000, B 0.000, C 0.000 }
gfCNCPoint2[28680] = {X 295.3508, Y 45.9791, Z -3.8333, A 0.000, B 0.000, C 0.000 }
gfCNCPoint2[28681] = {X 295.0254, Y 46.9091, Z -3.8333, A 0.000, B 0.000, C 0.000 }
gfCNCPoint2[28682] = {X 294.5012, Y 47.7434, Z -3.8333, A 0.000, B 0.000, C 0.000 }
gfCNCPoint2[28683] = {X 293.8045, Y 48.4401, Z -3.8333, A 0.000, B 0.000, C 0.000 }
gfCNCPoint2[28684] = {X 292.9702, Y 48.9643, Z -3.8333, A 0.000, B 0.000, C 0.000 }
gfCNCPoint2[28685] = {X 292.0402, Y 49.2897, Z -3.8333, A 0.000, B 0.000, C 0.000 }
gfCNCPoint2[28686] = {X 291.0611, Y 49.4000, Z -3.8333, A 0.000, B 0.000, C 0.000 }
gfCNCPoint2[28687] = {X 284.6177, Y 49.4000, Z -3.8333, A 0.000, B 0.000, C 0.000 }
gfCNCPoint2[28688] = {X 283.6386, Y 49.2897, Z -3.8333, A 0.000, B 0.000, C 0.000 }
gfCNCPoint2[28689] = {X 282.7086, Y 48.9643, Z -3.8333, A 0.000, B 0.000, C 0.000 }
gfCNCPoint2[28690] = {X 281.8743, Y 48.4400, Z -3.8333, A 0.000, B 0.000, C 0.000 }
gfCNCPoint2[28691] = {X 281.1776, Y 47.7433, Z -3.8333, A 0.000, B 0.000, C 0.000 }
gfCNCPoint2[28692] = {X 280.6534, Y 46.9091, Z -3.8333, A 0.000, B 0.000, C 0.000 }
gfCNCPoint2[28693] = {X 280.3280, Y 45.9791, Z -3.8333, A 0.000, B 0.000, C 0.000 }
gfCNCPoint2[28694] = {X 280.2177, Y 45.0000, Z -3.8333, A 0.000, B 0.000, C 0.000 }
gfCNCPoint2[28695] = {X 280.2177, Y 44.2067, Z -3.8333, A 0.000, B 0.000, C 0.000 }
gfCNCPoint2[28696] = {X 280.3226, Y 43.2698, Z -3.8333, A 0.000, B 0.000, C 0.000 }
gfCNCPoint2[28697] = {X 280.6226, Y 42.3759, Z -3.8333, A 0.000, B 0.000, C 0.000 }
gfCNCPoint2[28698] = {X 281.1041, Y 41.5654, Z -3.8333, A 0.000, B 0.000, C 0.000 }
gfCNCPoint2[28699] = {X 281.7456, Y 40.8744, Z -3.8333, A 0.000, B 0.000, C 0.000 }
gfCNCPoint2[28700] = {X 281.7452, Y 16.3110, Z -3.8333, A 0.000, B 0.000, C 0.000 }
gfCNCPoint2[28701] = {X 281.1006, Y 15.6219, Z -3.8333, A 0.000, B 0.000, C 0.000 }
gfCNCPoint2[28702] = {X 280.6177, Y 14.8112, Z -3.8333, A 0.000, B 0.000, C 0.000 }
gfCNCPoint2[28703] = {X 280.3188, Y 13.9161, Z -3.8333, A 0.000, B 0.000, C 0.000 }
gfCNCPoint2[28704] = {X 280.2177, Y 12.9779, Z -3.8333, A 0.000, B 0.000, C 0.000 }
gfCNCPoint2[28705] = {X 280.2177, Y 12.1868, Z -3.8333, A 0.000, B 0.000, C 0.000 }
gfCNCPoint2[28706] = {X 280.3280, Y 11.2077, Z -3.8333, A 0.000, B 0.000, C 0.000 }
gfCNCPoint2[28707] = {X 280.6534, Y 10.2777, Z -3.8333, A 0.000, B 0.000, C 0.000 }
gfCNCPoint2[28708] = {X 281.1776, Y 9.4435, Z -3.8333, A 0.000, B 0.000, C 0.000 }
gfCNCPoint2[28709] = {X 281.8743, Y 8.7468, Z -3.8333, A 0.000, B 0.000, C 0.000 }
gfCNCPoint2[28710] = {X 282.7086, Y 8.2226, Z -3.8333, A 0.000, B 0.000, C 0.000 }
gfCNCPoint2[28711] = {X 283.6386, Y 7.8971, Z -3.8333, A 0.000, B 0.000, C 0.000 }
gfCNCPoint2[28712] = {X 284.6177, Y 7.7868, Z -3.8333, A 0.000, B 0.000, C 0.000 }
gfCNCPoint2[28713] = {X 291.0611, Y 7.7868, Z -3.8333, A 0.000, B 0.000, C 0.000 }
gfCNCPoint2[28714] = {X 292.0402, Y 7.8971, Z -3.8333, A 0.000, B 0.000, C 0.000 }
gfCNCPoint2[28715] = {X 292.9702, Y 8.2226, Z -3.8333, A 0.000, B 0.000, C 0.000 }
gfCNCPoint2[28716] = {X 293.8045, Y 8.7468, Z -3.8333, A 0.000, B 0.000, C 0.000 }
gfCNCPoint2[28717] = {X 294.5012, Y 9.4435, Z -3.8333, A 0.000, B 0.000, C 0.000 }
gfCNCPoint2[28718] = {X 295.0254, Y 10.2777, Z -3.8333, A 0.000, B 0.000, C 0.000 }
gfCNCPoint2[28719] = {X 295.3508, Y 11.2077, Z -3.8333, A 0.000, B 0.000, C 0.000 }
gfCNCPoint2[28720] = {X 295.4611, Y 12.1868, Z -3.8333, A 0.000, B 0.000, C 0.000 }
gfCNCPoint2[28721] = {X 295.4609, Y 13.0233, Z -3.8333, A 0.000, B 0.000, C 0.000 }
gfCNCPoint2[28722] = {X 295.3526, Y 13.9495, Z -3.8333, A 0.000, B 0.000, C 0.000 }
gfCNCPoint2[28723] = {X 295.0515, Y 14.8320, Z -3.8333, A 0.000, B 0.000, C 0.000 }
gfCNCPoint2[28724] = {X 294.5712, Y 15.6312, Z -3.8333, A 0.000, B 0.000, C 0.000 }
gfCNCPoint2[28725] = {X 293.9333, Y 16.3113, Z -3.8333, A 0.000, B 0.000, C 0.000 }
gfCNCPoint2[28726] = {X 293.9344, Y 22.1165, Z -3.8333, A 0.000, B 0.000, C 0.000 }
gfCNCPoint2[28727] = {X 302.6792, Y 22.1165, Z -3.8333, A 0.000, B 0.000, C 0.000 }
gfCNCPoint2[28728] = {X 302.6797, Y 16.3110, Z -3.8333, A 0.000, B 0.000, C 0.000 }
gfCNCPoint2[28729] = {X 302.0351, Y 15.6218, Z -3.8333, A 0.000, B 0.000, C 0.000 }
gfCNCPoint2[28730] = {X 301.5523, Y 14.8111, Z -3.8333, A 0.000, B 0.000, C 0.000 }
gfCNCPoint2[28731] = {X 301.2534, Y 13.9161, Z -3.8333, A 0.000, B 0.000, C 0.000 }
gfCNCPoint2[28732] = {X 301.1523, Y 12.9779, Z -3.8333, A 0.000, B 0.000, C 0.000 }
gfCNCPoint2[28733] = {X 301.1523, Y 12.1868, Z -3.8333, A 0.000, B 0.000, C 0.000 }
gfCNCPoint2[28734] = {X 301.2626, Y 11.2077, Z -3.8333, A 0.000, B 0.000, C 0.000 }
gfCNCPoint2[28735] = {X 301.5880, Y 10.2777, Z -3.8333, A 0.000, B 0.000, C 0.000 }
gfCNCPoint2[28736] = {X 302.1122, Y 9.4435, Z -3.8333, A 0.000, B 0.000, C 0.000 }
gfCNCPoint2[28737] = {X 302.8089, Y 8.7468, Z -3.8333, A 0.000, B 0.000, C 0.000 }
gfCNCPoint2[28738] = {X 303.6432, Y 8.2226, Z -3.8333, A 0.000, B 0.000, C 0.000 }
gfCNCPoint2[28739] = {X 304.5732, Y 7.8971, Z -3.8333, A 0.000, B 0.000, C 0.000 }
gfCNCPoint2[28740] = {X 305.5523, Y 7.7868, Z -3.8333, A 0.000, B 0.000, C 0.000 }
gfCNCPoint2[28741] = {X 311.9957, Y 7.7868, Z -3.8333, A 0.000, B 0.000, C 0.000 }
gfCNCPoint2[28742] = {X 312.9748, Y 7.8971, Z -3.8333, A 0.000, B 0.000, C 0.000 }
gfCNCPoint2[28743] = {X 313.9048, Y 8.2226, Z -3.8333, A 0.000, B 0.000, C 0.000 }
gfCNCPoint2[28744] = {X 314.7391, Y 8.7468, Z -3.8333, A 0.000, B 0.000, C 0.000 }
gfCNCPoint2[28745] = {X 315.4358, Y 9.4435, Z -3.8333, A 0.000, B 0.000, C 0.000 }
gfCNCPoint2[28746] = {X 315.9600, Y 10.2777, Z -3.8333, A 0.000, B 0.000, C 0.000 }
gfCNCPoint2[28747] = {X 316.2854, Y 11.2077, Z -3.8333, A 0.000, B 0.000, C 0.000 }
gfCNCPoint2[28748] = {X 316.3957, Y 12.1868, Z -3.8333, A 0.000, B 0.000, C 0.000 }
gfCNCPoint2[28749] = {X 316.3955, Y 13.0233, Z -3.8333, A 0.000, B 0.000, C 0.000 }
gfCNCPoint2[28750] = {X 316.2872, Y 13.9494, Z -3.8333, A 0.000, B 0.000, C 0.000 }
gfCNCPoint2[28751] = {X 315.9861, Y 14.8319, Z -3.8333, A 0.000, B 0.000, C 0.000 }
gfCNCPoint2[28752] = {X 315.5059, Y 15.6311, Z -3.8333, A 0.000, B 0.000, C 0.000 }
gfCNCPoint2[28753] = {X 314.8680, Y 16.3112, Z -3.8333, A 0.000, B 0.000, C 0.000 }
gfCNCPoint2[28754] = {X 314.8678, Y 40.8754, Z -3.8333, A 0.000, B 0.000, C 0.000 }
gfCNCPoint2[28755] = {X 315.5126, Y 41.5646, Z -3.8333, A 0.000, B 0.000, C 0.000 }
gfCNCPoint2[28756] = {X 315.9956, Y 42.3754, Z -3.8333, A 0.000, B 0.000, C 0.000 }
gfCNCPoint2[28757] = {X 316.2945, Y 43.2706, Z -3.8333, A 0.000, B 0.000, C 0.000 }
gfCNCPoint2[28758] = {X 316.3957, Y 44.2089, Z -3.8333, A 0.000, B 0.000, C 0.000 }
gfCNCPoint2[28759] = {X 316.3957, Y 45.0000, Z -3.8333, A 0.000, B 0.000, C 0.000 }
gfCNCPoint2[28760] = {X 316.3190, Y 45.8182, Z -3.8333, A 0.000, B 0.000, C 0.000 }
gfCNCPoint2[28761] = {X 316.0914, Y 46.6079, Z -3.8333, A 0.000, B 0.000, C 0.000 }
gfCNCPoint2[28762] = {X 315.7209, Y 47.3415, Z -3.8333, A 0.000, B 0.000, C 0.000 }
gfCNCPoint2[28763] = {X 315.2205, Y 47.9934, Z -3.8333, A 0.000, B 0.000, C 0.000 }
gfCNCPoint2[28764] = {X 315.5723, Y 48.3200, Z -3.8333, A 0.000, B 0.000, C 0.000 }
